                  
END_PROGRAM

PROGRAM prg_Hmi_FrameMiniPCMenu
  VAR
    iSelectionFrameMiniPCMenu : INT;
    xTB_Home : BOOL;
  END_VAR

                    IF xTB_Home THEN
	xTB_Home := FALSE;
	iSelectionFrameMiniPCMenu := 0;
END_IF
                  
END_PROGRAM

PROGRAM prg_Hmi_ManagerMiniPC
  VAR
    sDescriptionBar : STRING(255) := 'Stato Gestore CubeOS:';
    sStatusMessage : STRING(255);
  END_VAR

                    // IF visuElems.CURRENTLANGUAGE = 'it' THEN
// 	sDescriptionBar := 'Gestore MiniPC:';
// ELSE
// 	sDescriptionBar := 'MiniPC manager:';
// END_IF

// sStatusMessage := GVL.g_PM_HMI_StatusMessages.sMiniPCManager;
                  
END_PROGRAM

PROGRAM prg_Hmi_InterfaceSetting
  VAR
    sDescriptionBar : STRING(255) := 'Stato impostazioni:';
    sStatusMessage : STRING(255);
  END_VAR

                    
                  
END_PROGRAM

PROGRAM prg_Hmi_RobotMenu
  VAR
    sDescriptionBar : STRING(255) := 'Stato Robot:';
    sStatusMessage : STRING(255);
    xTB_Refresh : BOOL;
    xDIS_Refresh : BOOL;
    sWebServerURL : STRING(255) := 'http://192.168.1.232:3000';
    xShowWebServerPage : BOOL := TRUE;
    sTestImageBitmap : STRING(255) := '/home/andrea/temp/history/detection_2023-03-31-09:36:17.png';
  END_VAR

                    xDIS_Refresh := xShowWebServerPage;
IF xTB_Refresh THEN
	xTB_Refresh := FALSE;
	xShowWebServerPage := TRUE;
END_IF
                  
END_PROGRAM

PROGRAM prg_Hmi_FrameRobotMenu
  VAR
    iSelectionFrameRobotMenu : INT;
    xTB_Home : BOOL;
  END_VAR

                    IF xTB_Home THEN
	xTB_Home := FALSE;
	iSelectionFrameRobotMenu := 0;
END_IF
                  
END_PROGRAM

PROGRAM prg_Hmi_ErrorFrame
  VAR
    iSelectionFrame : INT;
    sStatusMessage : STRING(255);
    sDescriptionBar : STRING(255);
  END_VAR

                    
                  
END_PROGRAM

PROGRAM prg_Hmi_Application
  VAR
    ROSInterface_01 : ros_interface_struct_t;
    xTB_Run_01 : BOOL;
    xDIS_Run_01 : BOOL;
    eROSProcessState_01 : process_code_enum_t;
    ROSInterface_02 : ros_interface_struct_t;
    xTB_Run_02 : BOOL;
    xDIS_Run_02 : BOOL;
    eROSProcessState_02 : process_code_enum_t;
    diProcessCode_01 : DINT;
    dwColorProcessState_01 : DWORD;
    eProcessState_01 : process_code_enum_t;
    dwFontColorID_01 : DWORD;
    diProcessCode_02 : DINT;
    dwColorProcessState_02 : DWORD;
    eProcessState_02 : process_code_enum_t;
    dwFontColorID_02 : DWORD;
    eDoosanRobotState : doosan_robot_state_enum_t;
    dwColorDoosanState : DWORD;
    xDIS_Run : BOOL;
    eDoosanRobotState_2 : doosan_robot_state_enum_t;
    dwColorDoosanState_2 : DWORD;
    xCommunicationError_2 : BOOL;
    xCommunicationError : BOOL;
    xINVIS_CommErr : BOOL;
    xDangerBlinkRed : BOOL;
    xEnableDangerBlinking : BOOL;
    xDangerBlinkRed_2 : BOOL;
    xINVIS_CommErr_2 : BOOL;
    sDescriptionBar : STRING(255) := 'Stato applicazione:';
    sStatusMessage : STRING(255);
  END_VAR

                    // IF visuElems.CURRENTLANGUAGE = 'it' THEN

ROSInterface_01 := prgROS.ROSInterface_01;
xTB_Run_01 := TO_BOOL(ROSInterface_01.Codesys2ROS.Published.run);
eROSProcessState_01 := ROSInterface_01.ROS2Codesys.eProcessState;
(*--------------------------------*)
ROSInterface_02 := prgROS.ROSInterface_02;
xTB_Run_02 := TO_BOOL(ROSInterface_02.Codesys2ROS.Published.run);
eROSProcessState_02 := ROSInterface_02.ROS2Codesys.eProcessState;

(*======================================================*)
diProcessCode_01 := prgROS.ROSInterface_01.ROS2Codesys.Subscripted.process_code;
eProcessState_01 := prgROS.ROSInterface_01.ROS2Codesys.eProcessState;

IF diProcessCode_01 < 0 THEN
	dwColorProcessState_01 := GVL_Constants.gc_dwRed;
ELSE
	dwColorProcessState_01 := GVL_Constants.gc_dwWhite;
END_IF

CASE eProcessState_01 OF
	process_code_enum_t.pcode_Error:
		dwFontColorID_01 := GVL_Constants.gc_dwRed;
	ELSE
		dwFontColorID_01 := GVL_Constants.gc_dwWhite;
END_CASE
(*======================================================*)
diProcessCode_02 := prgROS.ROSInterface_02.ROS2Codesys.Subscripted.process_code;
eProcessState_02 := prgROS.ROSInterface_02.ROS2Codesys.eProcessState;

IF diProcessCode_02 < 0 THEN
	dwColorProcessState_02 := GVL_Constants.gc_dwRed;
ELSE
	dwColorProcessState_02 := GVL_Constants.gc_dwWhite;
END_IF

CASE eProcessState_02 OF
	process_code_enum_t.pcode_Error:
		dwFontColorID_02 := GVL_Constants.gc_dwRed;
	ELSE
		dwFontColorID_02 := GVL_Constants.gc_dwWhite;
END_CASE

(**)

eDoosanRobotState := prgEIPMapping.DoosanState.eRobotState; //12/01/2023
CASE eDoosanRobotState OF
	doosan_robot_state_enum_t.EmergencyStop, doosan_robot_state_enum_t.SafeOff, doosan_robot_state_enum_t.BackdriveHold:
		dwColorDoosanState := GVL_Constants.gc_dwRed;
	doosan_robot_state_enum_t.StandaloneRunning:
		dwColorDoosanState := GVL_Constants.gc_dwGreen;
	ELSE
		dwColorDoosanState := GVL_Constants.gc_dwWhite;
END_CASE

xCommunicationError := prgEIPMapping.xCommunicationError;
IF xCommunicationError THEN
	xDangerBlinkRed := xEnableDangerBlinking AND prg_HMI_MainFrame.METH_GetBlinkSync_Slow();
ELSE
	xDangerBlinkRed := FALSE;
END_IF
IF xCommunicationError THEN
	xINVIS_CommErr := NOT prg_HMI_MainFrame.METH_GetBlinkSync_Fast();
ELSE
	xINVIS_CommErr := TRUE;
END_IF
// xDIS_Run := 
// 	(
// 		eDoosanRobotState = doosan_robot_state_enum_t.EmergencyStop 
// 		OR eDoosanRobotState = doosan_robot_state_enum_t.SafeOff 
// 		OR eDoosanRobotState = doosan_robot_state_enum_t.BackdriveHold
// 		OR prg_Hmi_RobotControl.eAdapterState <> IoDrvEtherNetIP.DEVICE_STATE.RUNNING
// 	) AND NOT METH_IsGazelle()
// ;

eDoosanRobotState_2 := prgEIPMapping.DoosanState_2.eRobotState; //12/01/2023
CASE eDoosanRobotState_2 OF
	doosan_robot_state_enum_t.EmergencyStop, doosan_robot_state_enum_t.SafeOff, doosan_robot_state_enum_t.BackdriveHold:
		dwColorDoosanState_2 := GVL_Constants.gc_dwRed;
	doosan_robot_state_enum_t.StandaloneRunning:
		dwColorDoosanState_2 := GVL_Constants.gc_dwGreen;
	ELSE
		dwColorDoosanState_2 := GVL_Constants.gc_dwWhite;
END_CASE

xCommunicationError_2 := prgEIPMapping.xCommunicationError_2;
IF xCommunicationError_2 THEN
	xDangerBlinkRed_2 := xEnableDangerBlinking AND prg_HMI_MainFrame.METH_GetBlinkSync_Slow();
ELSE
	xDangerBlinkRed_2 := FALSE;
END_IF
IF xCommunicationError_2 THEN
	xINVIS_CommErr_2 := NOT prg_HMI_MainFrame.METH_GetBlinkSync_Fast();
ELSE
	xINVIS_CommErr_2 := TRUE;
END_IF

                  

METHOD METH_IsGazelle : BOOL
                          METH_IsGazelle := prgMain.sHostName = 'gazelle';
                        
END_METHOD

METHOD METH_ToggleRun_01 : BOOL
  VAR
    xCurrentValue : BOOL;
    xVal : BOOL;
  END_VAR
                          xCurrentValue := TO_BOOL(prgROS.ROSInterface_01.Codesys2ROS.Published.run);
xVal := prgROS.METH_SetRun_01(xValue := NOT xCurrentValue);

METH_ToggleRun_01 := xVal;
                        
END_METHOD

METHOD METH_ToggleRun_02 : BOOL
  VAR
    xCurrentValue : BOOL;
    xVal : BOOL;
  END_VAR
                          xCurrentValue := TO_BOOL(prgROS.ROSInterface_02.Codesys2ROS.Published.run);
xVal := prgROS.METH_SetRun_02(xValue := NOT xCurrentValue);

METH_ToggleRun_02 := xVal;
                        
END_METHOD
END_PROGRAM

(* Implicitly generated code : DO NOT EDIT *)
{attribute 'check_bounds'}
{attribute 'no_check'}
FUNCTION CheckBounds : DINT
  VAR_INPUT
    index : DINT;
    lower : DINT;
    upper : DINT;
  END_VAR

                    // Implicitly generated code: Only an implementation suggestion
IF  index < lower THEN
	CheckBounds := lower;
ELSIF  index > upper THEN
	CheckBounds := upper;
ELSE  
	CheckBounds := index;
END_IF

(*It is also possible to set a breakpoint, log messages or e.g. to halt on an exception:
Add CmpApp.library, SysExcept.library and SysTypes2_Itf as newest.
Declaration:
VAR
    _pApp : POINTER TO CmpApp.APPLICATION;
    _result   : SysTypes.RTS_IEC_RESULT;
END_VAR

Implementation:
_pApp := AppGetCurrent(pResult:=_result);
IF  index < lower THEN
        CheckBounds := lower;
        IF _pApp <> 0 THEN
                AppGenerateException(pApp:=_pApp, ulException:=RtsExceptions.RTSEXCPT_ARRAYBOUNDS);
        END_IF
ELSIF  index > upper THEN
        CheckBounds := upper;
        IF _pApp <> 0 THEN
                AppGenerateException(pApp:=_pApp,   ulException:=RtsExceptions.RTSEXCPT_ARRAYBOUNDS);
        END_IF
ELSE  
        CheckBounds := index;
END_IF
*)

                  
END_FUNCTION

PROGRAM prgLinuxCommand
  VAR
    xTB_LinuxCommandTest : BOOL;
    xTB_NodeList : BOOL;
    diProcessExecuteResult : DINT;
    RTS_Result : SysProcess.RTS_IEC_RESULT;
    sCommand : STRING(255) := 'sudo pwd';
    sStdOutBuffer : STRING(1000);
    udiSizeStdOutBuffer : UDINT;
    iCounterFailure : INT;
    iCounterSuccess : INT;
    sLastStdOutResult : STRING(1000);
    sErrorMessage : STRING;
    xwCopySize : __XWORD;
    sPythonFile_Echo : STRING := 'echo.py';
    sPythonCommand_Echo : STRING(255) := 'CONCAT(c_sPythonExecute, sPythonFile_Echo)';
    sDestFullPath_Echo : STRING(255);
    sSourceFullPath_Echo : STRING(255);
    sBashFile_DockerActivate : STRING := 'launch_docker.sh';
    sBashCommand_DockerActivate : STRING(255) := 'CONCAT(c_sBashExecute, sBashFile_DockerActivate)';
    sDestFullPath_DockerActivate : STRING(255);
    sSourceFullPath_DockerActivate : STRING(255);
    sBashFile_RobinActivate : STRING := 'launch_remote_robin.sh';
    sBashCommand_RobinActivate : STRING(255) := 'CONCAT(c_sBashExecute, sBashFile_RobinActivate)';
    sDestFullPath_RobinActivate : STRING(255);
    sSourceFullPath_RobinActivate : STRING(255);
    xTB_ActivateDocker : BOOL;
    xTB_ActivateRobin : BOOL;
    sTestCommand : STRING(255) := 'sudo roscore';
    xTB_ShutdownMiniPC : BOOL;
    xDIS_Command : BOOL;
    xTB_RebootMiniPC : BOOL;
    xTB_StartDocker : BOOL;
    xTB_KillBehaviorTree : BOOL;
    xTB_StartBehaviorTree : BOOL;
    xTB_StopDocker : BOOL;
    xTB_ListDockers : BOOL;
    xListContainers : BOOL;
    sContainersAlive : STRING(1000);
    xTB_KillBoxDetection : BOOL;
    xTB_StartBoxDetection : BOOL;
    xTB_ReadFile : BOOL;
    RTS_FileCloseResult : RTS_IEC_RESULT;
    xListNodes : BOOL;
    sNodesAlive : STRING(255);
    TON_NodeList : TON;
    xTB_NodeListStartNode : BOOL;
    tTimeStart : TIME := TIME#3s0ms;
    TON_NodeListPolling : TON;
    xIsDockerDoosanStarted : BOOL;
    tPollingNodes : TIME := TIME#10s0ms;
    xTB_StartDoosanControl : BOOL;
    xTB_KillDoosanControl : BOOL;
    xTB_StartDoosanMover : BOOL;
    xTB_KillDoosanMover : BOOL;
    xIsDoosanControlStarted : BOOL;
    xIsDoosanMoverStarted : BOOL;
    xIsBoxRecognitionStarted : BOOL;
    xIsBehaviorStarted : BOOL;
    tPollingDocker : TIME := TIME#30s0ms;
    TON_DockerListPolling : TON;
    iStepStartAll : INT;
    xTB_StartAllNodes : BOOL;
    xNodeStartRequested : BOOL;
    xAllNodesDown : BOOL;  (* xTB_StopAllNodes: BOOL; *)
    xAllNodesAreUp : BOOL;
    xTB_START_DOOSAN : BOOL;
    xTB_STOP : BOOL;
    xTB_RECOVERY_TOOL_EMPTY : BOOL;
    xEnableListing : BOOL;
    xTB_RECOVERY_TOOL_BUNDLE : BOOL;
    xTB_RECOVERY_TOOL_STOP : BOOL;
    sCurrentDockerComposePath : STRING;
    xTB_START_BT01 : BOOL;
    xTB_START_BT02 : BOOL;
    xTB_STOP_BT01 : BOOL;
    xTB_STOP_BT02 : BOOL;
    xIsDockerBTStarted : BOOL;
    xIsDockerBTStarted01 : BOOL;
    xIsDockerBTStarted02 : BOOL;
  END_VAR
  VAR CONSTANT
    c_sDestPath : STRING := '/var/opt/codesys/';
    c_sSourcePath : STRING := '/var/opt/codesys/PlcLogic/Application/';
    c_sPythonExecute : STRING := 'sudo python ';
    c_sBashExecute : STRING := './';
    c_sDockerName : STRING := 'src-doosan';  (* philip_development //philip_devel-v2 //philip_development *)
    c_sDockerNameBT : STRING := 'src-behavior_tree';
    c_sDockerNameBT01 : STRING := 'src-behavior_tree1';
    c_sDockerNameBT02 : STRING := 'src-behavior_tree2';
    c_sDockerActivateFile : STRING := 'launch_docker.sh';
    c_sDockerComposePath_Gazelle : STRING := '/home/nicola/ros/philip_ws/src/';  (* 05/12/2022 *)
    c_sDockerComposePath_Cincoze : STRING := '/home/sysdesign/ros/philip_ws/src/';  (* 05/12/2022 *)
    c_sDockerComposePath_Esaware : STRING := '/home/sysdesign/ros/pallcube_ws/src/';  (* 05/12/2022 *)
  END_VAR

                    (*=======================================================*)
// MINI PC
ACT_MiniPC();

(*--------------------------------*)
// dockker list
ACT_DockerList();
(*--------------------------------*)
// docker compose command
ACT_Start();

ACT_Stop();

(*--------------------------------*)
// flags
xIsDoosanControlStarted := FIND(sNodesAlive, 'dsr01h2017') > 0;
xIsDoosanMoverStarted := FIND(sNodesAlive, 'doosan_mover') > 0;
xIsBoxRecognitionStarted := FIND(sNodesAlive, 'box_recognition') > 0;
xIsBehaviorStarted := FIND(sNodesAlive, 'behavior_tree') > 0;
(*--------------------------------*)
xDIS_Command := FALSE;
IF xTB_LinuxCommandTest THEN
	xTB_LinuxCommandTest := FALSE;
	xDIS_Command := TRUE; //06/12/2022
	
	sCommand := sTestCommand;
// 	sCommand := sPythonCommand_Echo;
	
	sErrorMessage := '';
	udiSizeStdOutBuffer := TO_UDINT(XSIZEOF(sStdOutBuffer));
	SysMem.SysMemSet(pDest := ADR(sStdOutBuffer), udiCount := XSIZEOF(sStdOutBuffer), udiValue := 0);
	
	diProcessExecuteResult := SysProcess.SysProcessExecuteCommand2(
		pszCommand := sCommand,
		pResult := ADR(RTS_Result),
		pszStdOut := sStdOutBuffer,
		udiStdOutLen := udiSizeStdOutBuffer
	);
	
	IF RTS_Result = CmpErrors.Errors.ERR_OK THEN
		iCounterSuccess := (iCounterSuccess + 1) MOD 16#7FFF;
		IF diProcessExecuteResult > 0 THEN // there is something to read
			sLastStdOutResult := sStdOutBuffer;
		END_IF
		IF xListContainers THEN
			xListContainers := FALSE;
			sContainersAlive := sStdOutBuffer;
		END_IF
		IF xListNodes THEN
			xListNodes := FALSE;
			sNodesAlive := sStdOutBuffer;
		END_IF
	ELSE
		sErrorMessage := METH_GetErrorMessage(udiResult := RTS_Result);
		iCounterFailure := (iCounterFailure + 1) MOD 16#7FFF;
		IF xListNodes THEN
			xListNodes := FALSE;
			sNodesAlive := '';
		END_IF
	END_IF
	
	xDIS_Command := FALSE; //06/12/2022
END_IF
(*=======================================================*)
                  

ACTION ACT_MiniPC:
                        IF xTB_ShutdownMiniPC OR GVL.g_xShutdownMiniPC THEN
	GVL.g_xShutdownMiniPC := FALSE;
	xTB_ShutdownMiniPC := FALSE;
	sTestCommand := 'sudo shutdown -h now';
	xTB_LinuxCommandTest := TRUE;
END_IF
IF xTB_RebootMiniPC THEN
	xTB_RebootMiniPC := FALSE;
	sTestCommand := 'sudo reboot';
	xTB_LinuxCommandTest := TRUE;
END_IF
                      
END_ACTION

ACTION ACT_DockerList:
                        // DOCKER list
TON_DockerListPolling(IN := xEnableListing, PT := tPollingDocker);
IF TON_DockerListPolling.Q THEN
	TON_DockerListPolling(IN := FALSE);
	xTB_ListDockers := TRUE;
END_IF
IF xTB_ListDockers OR GVL.g_xListDockers THEN
	GVL.g_xListDockers := FALSE;
	xTB_ListDockers := FALSE;
	sTestCommand := 'docker container ls';
	xTB_LinuxCommandTest := TRUE;
	xListContainers := TRUE;
END_IF

xIsDockerDoosanStarted := STU.StrFindA(pst1 := ADR(sContainersAlive), pst2 := ADR(c_sDockerName), uiSearchStart := 0) > 0;
xIsDockerBTStarted := STU.StrFindA(pst1 := ADR(sContainersAlive), pst2 := ADR(c_sDockerNameBT), uiSearchStart := 0) > 0;
xIsDockerBTStarted01 := STU.StrFindA(pst1 := ADR(sContainersAlive), pst2 := ADR(c_sDockerNameBT01), uiSearchStart := 0) > 0;
xIsDockerBTStarted02 := STU.StrFindA(pst1 := ADR(sContainersAlive), pst2 := ADR(c_sDockerNameBT02), uiSearchStart := 0) > 0;
TON_NodeListPolling(IN := xIsDockerDoosanStarted AND xEnableListing, PT := tPollingNodes);
IF TON_NodeListPolling.Q THEN
	TON_NodeListPolling(IN := FALSE);
	xTB_NodeList := TRUE;
END_IF
(*===============================================*)
// LIST
IF xTB_NodeList THEN
	xTB_NodeList := FALSE;
// 	sTestCommand := './launch_docker.sh';
	sTestCommand := '';
// 	sTestCommand := 'docker exec ';
// 	sTestCommand := CONCAT(sTestCommand, c_sDockerName);
// 	sTestCommand := CONCAT(sTestCommand, ' bash -c $'source devel/setup.bash; rosnode list$'');
	sTestCommand := 'bash -c $'source /opt/ros/noetic/setup.bash; rosnode list$'';
	xTB_LinuxCommandTest := TRUE;
	xListNodes := TRUE;
END_IF
(*--------------------------------*)
                      
END_ACTION

ACTION ACT_Start:
                        // DOOSAN
IF xTB_START_DOOSAN OR GVL.g_xNODES_START THEN // START DOOSAN
	xTB_START_DOOSAN := FALSE;
	GVL.g_xNODES_START := FALSE;
	sTestCommand := '';
	sCurrentDockerComposePath := METH_GetDockerComposePath();
	sTestCommand := CONCAT('docker compose -f ', CONCAT(sCurrentDockerComposePath, 'docker-compose.yml up -d doosan'));
	// 		sTestCommand := 'docker compose -f /home/nicola/ros/philip_ws/src/docker-compose.devel.yml up -d';
	// 	sTestCommand := 'bash /home/sysdesign/philip.sh start';
	xTB_LinuxCommandTest := TRUE;
END_IF

// BT
IF xTB_START_BT01 THEN // START DOOSAN
	xTB_START_BT01 := FALSE;
	sTestCommand := '';
	sCurrentDockerComposePath := METH_GetDockerComposePath();
	sTestCommand := CONCAT('docker compose -f ', CONCAT(sCurrentDockerComposePath, 'docker-compose.yml up -d behavior_tree1'));
	// 		sTestCommand := 'docker compose -f /home/nicola/ros/philip_ws/src/docker-compose.devel.yml up -d';
	// 	sTestCommand := 'bash /home/sysdesign/philip.sh start';
	xTB_LinuxCommandTest := TRUE;
END_IF

IF xTB_START_BT02 THEN // START DOOSAN
	xTB_START_BT02 := FALSE;
	sTestCommand := '';
	sCurrentDockerComposePath := METH_GetDockerComposePath();
	sTestCommand := CONCAT('docker compose -f ', CONCAT(sCurrentDockerComposePath, 'docker-compose.yml up -d behavior_tree2'));
	// 		sTestCommand := 'docker compose -f /home/nicola/ros/philip_ws/src/docker-compose.devel.yml up -d';
	// 	sTestCommand := 'bash /home/sysdesign/philip.sh start';
	xTB_LinuxCommandTest := TRUE;
END_IF
                      
END_ACTION

ACTION ACT_Stop:
                        IF xTB_STOP OR GVL.g_xNODES_STOP THEN
	xTB_STOP := FALSE;
	GVL.g_xNODES_STOP := FALSE;
	sTestCommand := '';
	sCurrentDockerComposePath := METH_GetDockerComposePath();
	sTestCommand := CONCAT('docker compose -f ', CONCAT(sCurrentDockerComposePath, 'docker-compose.yml down')); //23/01/2023: perche non STOP?
	// 		sTestCommand := 'docker compose -f /home/nicola/ros/philip_ws/src/docker-compose.devel.yml down';
// 		sTestCommand := 'bash /home/sysdesign/philip.sh stop';
	xTB_LinuxCommandTest := TRUE;
END_IF


IF xTB_STOP_BT01 THEN // START DOOSAN
	xTB_STOP_BT01 := FALSE;
	sTestCommand := '';
	sCurrentDockerComposePath := METH_GetDockerComposePath();
	sTestCommand := CONCAT('docker compose -f ', CONCAT(sCurrentDockerComposePath, 'docker-compose.yml stop behavior_tree1'));
	// 		sTestCommand := 'docker compose -f /home/nicola/ros/philip_ws/src/docker-compose.devel.yml up -d';
	// 	sTestCommand := 'bash /home/sysdesign/philip.sh start';
	xTB_LinuxCommandTest := TRUE;
END_IF

IF xTB_STOP_BT02 THEN // START DOOSAN
	xTB_STOP_BT02 := FALSE;
	sTestCommand := '';
	sCurrentDockerComposePath := METH_GetDockerComposePath();
	sTestCommand := CONCAT('docker compose -f ', CONCAT(sCurrentDockerComposePath, 'docker-compose.yml stop behavior_tree2'));
	// 		sTestCommand := 'docker compose -f /home/nicola/ros/philip_ws/src/docker-compose.devel.yml up -d';
	// 	sTestCommand := 'bash /home/sysdesign/philip.sh start';
	xTB_LinuxCommandTest := TRUE;
END_IF
                      
END_ACTION

METHOD METH_GetErrorMessage : STRING(255)
  VAR_INPUT
    udiResult : SysProcess.RTS_IEC_RESULT;
  END_VAR
  VAR
    sRes : STRING(255);
  END_VAR
                          CASE udiResult OF
	CmpErrors.Errors.ERR_PARAMETER:
		sRes := 'Some null input parameter';
	CmpErrors.Errors.ERR_NO_ACCESS_RIGHTS:
		sRes := 'Not allowed';
	CmpErrors.Errors.ERR_FAILED:
		sRes := 'Internal error';
	ELSE
		sRes := 'Error';
END_CASE

METH_GetErrorMessage := sRes;
                        
END_METHOD

METHOD METH_GetDockerComposePath : STRING
  VAR
    sRes : STRING;
  END_VAR
                          IF prgMAIN.sHostName = 'gazelle' OR prgMAIN.sHostName = 'esaware' THEN
	sRes := c_sDockerComposePath_Esaware;
ELSE
	sRes := c_sDockerComposePath_Cincoze;
END_IF

METH_GetDockerComposePath := sRes;
                        
END_METHOD

METHOD METH_StartDoosanDocker
                          xTB_START_DOOSAN := TRUE;
                        
END_METHOD

METHOD METH_StartBT01
                          xTB_START_BT01 := TRUE;
                        
END_METHOD

METHOD METH_StartBT02
                          xTB_START_BT02 := TRUE;
                        
END_METHOD

METHOD METH_StopAllDockers
                          xTB_STOP := TRUE;
                        
END_METHOD

METHOD METH_ShutdownMiniPC
                          xTB_ShutdownMiniPC := TRUE;
                        
END_METHOD

METHOD METH_RebootMiniPC
                          xTB_RebootMiniPC := TRUE;
                        
END_METHOD

METHOD METH_ListDockers
                          xTB_ListDockers := TRUE;
                        
END_METHOD

METHOD METH_IsDockerDoosanActive : BOOL
                          METH_IsDockerDoosanActive := xIsDockerDoosanStarted;

                        
END_METHOD

METHOD METH_IsDockerBTActive : BOOL
                          METH_IsDockerBTActive := xIsDockerBTStarted;

                        
END_METHOD

METHOD METH_IsDockerBTActive_01 : BOOL
                          METH_IsDockerBTActive_01 := xIsDockerBTStarted01;

                        
END_METHOD

METHOD METH_IsDockerBTActive_02 : BOOL
                          METH_IsDockerBTActive_02 := xIsDockerBTStarted02;

                        
END_METHOD

METHOD METH_StopBT01
                          xTB_STOP_BT01 := TRUE;
                        
END_METHOD

METHOD METH_StopBT02
                          xTB_STOP_BT02 := TRUE;
                        
END_METHOD
END_PROGRAM

PROGRAM prgEIPMapping
  VAR
    bRobotState : BYTE;
    bRobotFlags : BYTE;
    DoosanState : doosan_state_struct_t;  (* 16/12/2022 *)
    xCommunicationError : BOOL;
    xAirAspriration : BOOL;
    bRobotState_2 : BYTE;
    bRobotFlags_2 : BYTE;
    DoosanState_2 : doosan_state_struct_t;  (* 16/12/2022 *)
    xCommunicationError_2 : BOOL;
    TON_Dead_2 : TON;
    Doosan_EIP : doosan_t;
    Doosan_EIP_2 : doosan_t;
    udiRobotState : UDINT;
    xErrorArea : BOOL;
    TON_Dead : TON;  (* eProposedDoosanArea : PM_areas_enum_t; *)
    tDead : TIME := TIME#5s0ms;
    xInit : BOOL := TRUE;
    pxTurnOn : POINTER TO BOOL;
    xEthercatError : BOOL;
    xStartDocker : BOOL;
    xRecoveryZoneError : BOOL;
    xInRecoveryZone : BOOL;
  END_VAR

                    // EIP mask inputs
IO_Variables.g_Doosan_EIP.Cartesian := Doosan_EIP.Cartesian;
IO_Variables.g_Doosan_EIP.Joints := Doosan_EIP.Joints;
IO_Variables.g_Doosan_EIP.InfoRobot := Doosan_EIP.InfoRobot;

// eProposedDoosanArea := METH_GetArea(xError => xErrorArea, xIsAlive => IO_Variables.g_Doosan_EIP.xIsAlive); //20/10/2022: is alive
// IF NOT xErrorArea THEN
// 	IO_Variables.g_eDoosanArea := eProposedDoosanArea;
// ELSE
// 	IO_Variables.g_eDoosanArea := PM_areas_enum_t.UnknownArea;
// END_IF

xInRecoveryZone := METH_GetJointsLimitDanger(xError => xRecoveryZoneError); //07/12/2022

// 20/10/2022: automatically turn on doosan if
IO_Variables.g_Doosan_EIP.xIsAlive := prg_Hmi_RobotControl.eAdapterState = IoDrvEtherNetIP.DEVICE_STATE.RUNNING;//20/10/2022
xCommunicationError := NOT IO_Variables.g_Doosan_EIP.xIsAlive;
TON_Dead(IN := NOT IO_Variables.g_Doosan_EIP.xIsAlive, PT := tDead); //20/10/2022
GVL.g_xDoosanMayBeOff := TON_Dead.Q; //20/10/2022

IO_Variables.g_Doosan_EIP_2.xIsAlive := prg_Hmi_RobotControl2.eAdapterState = IoDrvEtherNetIP.DEVICE_STATE.RUNNING;//20/10/2022
xCommunicationError_2 := NOT IO_Variables.g_Doosan_EIP_2.xIsAlive;
TON_Dead_2(IN := NOT IO_Variables.g_Doosan_EIP_2.xIsAlive, PT := tDead); //20/10/2022
GVL.g_xDoosanMayBeOff_2 := TON_Dead_2.Q; //20/10/2022
// xEthercatError := 
// 	(prgMain.eEthercatState <> DED.BUS_STATE.RUNNING
// 	OR prgMain.eEthercatError <> DED.ERROR.NO_ERROR)
// // 	AND prgMain.xEthercatDiagnosisAvail //07/12/2022: commentato
// ; //24/10/2022: controllo ethercat prima di mandare segnale
// IF xInit THEN  
// 	IF IO_Variables.g_Doosan_EIP.xIsAlive THEN//20/10/2022
// 		xInit := FALSE;
// 		xStartDocker := TRUE; //28/10/2022: at startup also start docker
// 	ELSE  
// 		IF GVL.g_xDoosanMayBeOff AND NOT xEthercatError THEN //24/10/2022 //20/10/2022 
// // 			pxTurnOn := ADR(prg_Hmi_Home.xTB_TurnDoosanON);
// // 			pxTurnOn^ := TRUE;
// 			prg_Hmi_Home.METH_AskForDoosanOn();
// 			xInit := FALSE;
// 			xStartDocker := TRUE; //28/10/2022: at startup also start docker
// 		END_IF
// 	END_IF
// ELSIF xStartDocker THEN //28/10/2022 starts docker at startup
// 	IF IO_Variables.g_Doosan_EIP.xIsAlive THEN
// 		GVL.g_xNODES_START := TRUE;
// 		xStartDocker := FALSE;
// 	END_IF
// END_IF
(*--------------------------------------------------------------*)
//16/12/2022: flag per capire se stato robot è quel che voglio
DoosanState.eRobotState := bRobotState;
DoosanState.xSO_ServoOn := bRobotFlags.0;
DoosanState.xSS_SafetyStopped := bRobotFlags.1;
DoosanState.xES_EmergencyStopped := bRobotFlags.2;
DoosanState.xDTPB_DirectTeachButtonPressed := bRobotFlags.3;
DoosanState.xPBP_PowerButtonPressed := bRobotFlags.4;

DoosanState_2.eRobotState := bRobotState_2;
DoosanState_2.xSO_ServoOn := bRobotFlags_2.0;
DoosanState_2.xSS_SafetyStopped := bRobotFlags_2.1;
DoosanState_2.xES_EmergencyStopped := bRobotFlags_2.2;
DoosanState_2.xDTPB_DirectTeachButtonPressed := bRobotFlags_2.3;
DoosanState_2.xPBP_PowerButtonPressed := bRobotFlags_2.4;



                  

(* This method proposes an area, but if more then one is found, then it throws an error *)
METHOD METH_GetArea : PM_areas_enum_t
  VAR_OUTPUT
    xError : BOOL;
    xIsAlive : BOOL;  (* 20/10/2022 *)
  END_VAR
  VAR
    eRes : PM_areas_enum_t;
    aHome_WindowX : ARRAY[0..1] OF REAL := [(-640.0 - 200), (-640.0 + 200.0)];
    aHome_WindowY : ARRAY[0..1] OF REAL := [(-210.0 - 200), (-210.0 + 200)];
    aHome_WindowZ : ARRAY[0..1] OF REAL := [700.0, 1100.0];
    xInHomeArea : BOOL;
    aLoadCube_WindowX : ARRAY[0..1] OF REAL := [0.0, 0.0];
    aLoadCube_WindowY : ARRAY[0..1] OF REAL := [0.0, 0.0];
    aLoadCube_WindowZ : ARRAY[0..1] OF REAL := [0.0, 0.0];
    xInLoadCubeArea : BOOL;
    aPallet_WindowX : ARRAY[0..1] OF REAL := [0.0, 0.0];
    aPallet_WindowY : ARRAY[0..1] OF REAL := [0.0, 0.0];
    aPallet_WindowZ : ARRAY[0..1] OF REAL := [0.0, 0.0];
    xInPalletArea : BOOL;
    aSenzani_WindowX : ARRAY[0..1] OF REAL := [0.0, 0.0];
    aSenzani_WindowY : ARRAY[0..1] OF REAL := [0.0, 0.0];
    aSenzani_WindowZ : ARRAY[0..1] OF REAL := [0.0, 0.0];
    xInSenzaniArea : BOOL;
    lrX : REAL;
    lrY : REAL;
    lrZ : REAL;
    lrA : REAL;
    lrB : REAL;
    lrC : REAL;
    xConflict : BOOL;
    xAllZero : BOOL;
    xAllZeroJoints : BOOL;
  END_VAR
                          lrX := IO_Variables.g_Doosan_EIP.Cartesian.x;
lrY := IO_Variables.g_Doosan_EIP.Cartesian.y;
lrZ := IO_Variables.g_Doosan_EIP.Cartesian.z;
lrA := IO_Variables.g_Doosan_EIP.Cartesian.A;
lrB := IO_Variables.g_Doosan_EIP.Cartesian.B;
lrC := IO_Variables.g_Doosan_EIP.Cartesian.C;

xAllZero := lrX = 0.0 AND lrY = 0.0 AND lrZ = 0.0 AND lrA = 0.0 AND lrB = 0.0 AND lrC = 0.0;
xAllZeroJoints := 
	IO_Variables.g_Doosan_EIP.Joints.j1 = 0.0
	AND IO_Variables.g_Doosan_EIP.Joints.j2 = 0.0
	AND IO_Variables.g_Doosan_EIP.Joints.j3 = 0.0
	AND IO_Variables.g_Doosan_EIP.Joints.j4 = 0.0
	AND IO_Variables.g_Doosan_EIP.Joints.j5 = 0.0
	AND IO_Variables.g_Doosan_EIP.Joints.j6 = 0.0
;

xInHomeArea := 
	(lrX >= aHome_WindowX[0] AND lrX <= aHome_WindowX[1])
	AND (lrY >= aHome_WindowY[0] AND lrY <= aHome_WindowY[1])
	AND (lrZ >= aHome_WindowZ[0] AND lrZ <= aHome_WindowZ[1])
;

// 13/01/2023:  in load cube area for turning off
aLoadCube_WindowX := aHome_WindowX;
aLoadCube_WindowY := aHome_WindowY;
aHome_WindowZ[0] := 200.0;
aHome_WindowZ[1] := aHome_WindowZ[0];
xInLoadCubeArea := 
	(lrX >= aLoadCube_WindowX[0] AND lrX <= aLoadCube_WindowX[1])
	AND (lrY >= aLoadCube_WindowY[0] AND lrY <= aLoadCube_WindowY[1])
	AND (lrZ >= aLoadCube_WindowZ[0] AND lrZ <= aLoadCube_WindowZ[1])
;

xInPalletArea := 
	(lrX >= aPallet_WindowX[0] AND lrX <= aPallet_WindowX[1])
	AND (lrY >= aPallet_WindowY[0] AND lrY <= aPallet_WindowY[1])
	AND (lrZ >= aPallet_WindowZ[0] AND lrZ <= aPallet_WindowZ[1])
;

xInSenzaniArea := 
	(lrX >= aSenzani_WindowX[0] AND lrX <= aSenzani_WindowX[1])
	AND (lrY >= aSenzani_WindowY[0] AND lrY <= aSenzani_WindowY[1])
	AND (lrZ >= aSenzani_WindowZ[0] AND lrZ <= aSenzani_WindowZ[1])
;

xConflict := TO_INT(xInHomeArea) + TO_INT(xInLoadCubeArea) + TO_INT(xInPalletArea) + TO_INT(xInSenzaniArea) > 1;

xError := xConflict OR xAllZero;

IF xInHomeArea THEN
	eRes := PM_areas_enum_t.HomeArea;
ELSIF xInLoadCubeArea THEN
	eRes := PM_areas_enum_t.LoadCubeArea;
ELSIF xInPalletArea THEN
	eRes := PM_areas_enum_t.PalletArea;
ELSIF xInSenzaniArea THEN
	eRes := PM_areas_enum_t.SenzaniArea;
ELSE
	eRes := PM_areas_enum_t.UnknownArea;
END_IF

xIsAlive := NOT (xAllZero AND xAllZeroJoints);

METH_GetArea := eRes;
                        
END_METHOD

(* This method proposes an area, but if more then one is found, then it throws an error *)
METHOD METH_GetJointsLimitDanger : BOOL
  VAR_OUTPUT
    xError : BOOL;
  END_VAR
  VAR
    xAllZeroJoints : BOOL;
    iInd : INT;
    iMaxInd : INT := 5;
    rJointVal : REAL;
    rAbsLimit : REAL;
    rTolerance : REAL;
    axJointsDanger : ARRAY[0..5] OF BOOL;
    xRes : BOOL;
  END_VAR
                          
xAllZeroJoints := 
	IO_Variables.g_Doosan_EIP.Joints.j1 = 0.0
	AND IO_Variables.g_Doosan_EIP.Joints.j2 = 0.0
	AND IO_Variables.g_Doosan_EIP.Joints.j3 = 0.0
	AND IO_Variables.g_Doosan_EIP.Joints.j4 = 0.0
	AND IO_Variables.g_Doosan_EIP.Joints.j5 = 0.0
	AND IO_Variables.g_Doosan_EIP.Joints.j6 = 0.0
;
FOR iInd := 0 TO iMaxInd DO
	CASE iInd OF
		0: 
			rJointVal := IO_Variables.g_Doosan_EIP.Joints.j1;
			rAbsLimit := TO_REAL(ABS(360.0));
		1:
			rJointVal := IO_Variables.g_Doosan_EIP.Joints.j2;
			rAbsLimit := TO_REAL(ABS(360.0));
		2:
			rJointVal := IO_Variables.g_Doosan_EIP.Joints.j2;
			rAbsLimit := TO_REAL(ABS(360.0));
		3:
			rJointVal := IO_Variables.g_Doosan_EIP.Joints.j2;
			rAbsLimit := TO_REAL(ABS(360.0));
		4:
			rJointVal := IO_Variables.g_Doosan_EIP.Joints.j2;
			rAbsLimit := TO_REAL(ABS(90.0));
		5:
			rJointVal := IO_Variables.g_Doosan_EIP.Joints.j2;
			rAbsLimit := TO_REAL(ABS(360.0));
	END_CASE
	axJointsDanger[iInd] := rJointVal <= -rAbsLimit OR rJointVal >= rAbsLimit;
	xRes := xRes OR axJointsDanger[iInd];
END_FOR


xError := xAllZeroJoints;

METH_GetJointsLimitDanger := xRes;
                        
END_METHOD

METHOD METH_IsDoosanServoOn : BOOL
  VAR_INPUT
    DoosanState : doosan_state_struct_t;
  END_VAR
                          METH_IsDoosanServoOn := DoosanState.xSO_ServoOn;
                        
END_METHOD

METHOD METH_IsDoosanReadyForManual : BOOL
  VAR_INPUT
    DoosanState : doosan_state_struct_t;
  END_VAR
                          METH_IsDoosanReadyForManual := DoosanState.eRobotState = doosan_robot_state_enum_t.ManualStandby;
                        
END_METHOD

METHOD METH_IsDoosanReadyForAuto : BOOL
  VAR_INPUT
    DoosanState : doosan_state_struct_t;
  END_VAR
                          METH_IsDoosanReadyForAuto := DoosanState.eRobotState = doosan_robot_state_enum_t.StandaloneStandby;
                        
END_METHOD

METHOD METH_IsDoosanSafeOff : BOOL
  VAR_INPUT
    DoosanState : doosan_state_struct_t;
  END_VAR
                          METH_IsDoosanSafeOff := DoosanState.eRobotState = doosan_robot_state_enum_t.SafeOff;
                        
END_METHOD

METHOD METH_IsDoosanTurnedOff : BOOL
  VAR_INPUT
    eAdapterState : IoDrvEtherNetIP.DEVICE_STATE;
  END_VAR
                          METH_IsDoosanTurnedOff := prg_Hmi_RobotControl.eAdapterState = IoDrvEtherNetIP.DEVICE_STATE.NOT_FOUND;
                        
END_METHOD
END_PROGRAM

PROGRAM prg_Hmi_AskedPose
  VAR
    xINVIS_JointsResults : BOOL := TRUE;
    xINVIS_CartResults : BOOL := TRUE;
    arValues : ARRAY[0..7] OF REAL;
    xTB_Convert : BOOL;
    diLengthValues : DINT;
    sValues : STRING(255);
    diInd : DINT;
    sCurrentValue : STRING(255);
    iStartPos : INT;
    iLength : INT;
    uiStartSearch : UINT;
    iFindINd : INT;
    iIndValues : INT;
    eInputType : pose_type_t;
    xDIS_EnableConversion : BOOL;
    iMinInputType : INT := ANY_TO_INT(pose_type_t.JointDegrees);
    iMaxInputType : INT := ANY_TO_INT(pose_type_t.Cart_m_quat);
    xConvertToJointRadians : BOOL;
    xConvertToJointDegrees : BOOL;
    xConvertFromZYZ : BOOL;
    xConvertFromRPY : BOOL;
    xConvertFromQuat : BOOL;
    iIndJoints : INT;
    xIgnoreCart : BOOL;
    udiAuxBufferSize : UDINT;
    sZYZ : STRING(255);
    rA : REAL;
    rB : REAL;
    rC : REAL;
    lrA : LREAL;
    lrB : LREAL;
    lrC : LREAL;
    sDescriptionBar : STRING(255);
    sStatusBar : STRING(255);
    sjAux : STRING;  (* - *)
    sStringJointPos : STRING;
    scAux : STRING;  (* - *)
    sStringCartPos : STRING;
    sQuaternion : STRING(255);
    lrRoll : LREAL;
    lrPitch : LREAL;
    lrYaw : LREAL;
    xToRPY : BOOL;
    rRoll : REAL;
    rPitch : REAL;
    rYaw : REAL;
    rXmm : REAL;
    rYmm : REAL;
    rZmm : REAL;
    sRPY : STRING(255);
    xIsRot : BOOL;
    arJointsInRadians : ARRAY[0..5] OF REAL;
    arJointsInDegrees : ARRAY[0..5] OF REAL;
    arCartZYZ : ARRAY[0..5] OF REAL;
    arCartQuat : ARRAY[0..5] OF REAL;
    arCartRPY : ARRAY[0..5] OF REAL;
    xTB_ParseString : BOOL;
    Set_IP : BOOL;
    ipDosan : ARRAY[0..3] OF BYTE;
    deinfo : IoDrvEtherNetIP.DEVICE_INFO;
    errorDE : IoDrvEtherNetIP.DED.ERROR;
    a_ipDoosan : ARRAY[0..3] OF ARRAY[0..3] OF STRING := [['192', '168', '1', '70'], 3([4('')])];
    iIndexIP : INT := 1;  (* -Default impostato sul Doosan *)
    rXMeters : REAL;
    rYMeters : REAL;
    rZMeters : REAL;
    rQW : REAL;
    rQX : REAL;
    rQY : REAL;
    rQZ : REAL;
    mR : SM3M.SMC_Matrix3;
    xComputeRotMat : BOOL;
    q : SM3M.SMC_Quat;
    quat : SM3M.SMC_Quat;
    sAux : STRING(255);
    iBufferSize : INT;
    sJointsInRadians : STRING(255);
    sJointsInDegrees : STRING(255);
  END_VAR

                    IF xTB_ParseString OR xTB_Convert THEN
	xINVIS_CartResults := TRUE;
	xINVIS_JointsResults := TRUE;
	xConvertToJointRadians := FALSE;
	xConvertToJointDegrees := FALSE;
	xConvertFromQuat := FALSE;
	xConvertFromRPY := FALSE;
	xConvertFromZYZ := FALSE;
	
	xTB_ParseString := FALSE;
	SysMem.SysMemSet(pDest := ADR(arValues), udiCount := XSIZEOF(arValues), udiValue := 0);
	diLengthValues := STU.StrLenA(pstData := ADR(sValues));
	diInd := 0;
	iStartPos := 0;
	iLength := 0;
	iIndValues := 0;
	WHILE diInd < diLengthValues DO
		sCurrentValue := '';
		uiStartSearch := TO_UINT(diInd);
		iFindInd := STU.StrCaseFindA(pst1 := ADR(sValues), pst2 := ADR(';'), uiSearchStart := uiStartSearch);
		IF iFindInd > 0 THEN
			IF diInd = 0 THEN // first value
				iStartPos := 1;
			ELSE
				iStartPos := TO_INT(diInd);
			END_IF
			iLength := iFindInd - iStartPos;
			
			STU.StrMidA(
				pstResult := ADR(sCurrentValue),
				uiResultBufferSize := TO_UINT(XSIZEOF(sCurrentValue)),
				pst := ADR(sValues),
				uiInputBufferSize := TO_UINT(XSIZEOF(sValues)),
				iPosition := iStartPos,
				iLength := iLength
			);
			arValues[iIndValues] := STRING_TO_REAL(sCurrentValue);
			iIndValues := iIndValues + 1;
			
			diInd := TO_DINT(iFindInd + 1);
		ELSE
			IF iStartPos > 0 THEN // last value (no ;)
				iStartPos := TO_INT(diInd);
				iLength := TO_INT(diLengthValues) + 1 - iStartPos;
				STU.StrMidA(
					pstResult := ADR(sCurrentValue),
					uiResultBufferSize := TO_UINT(XSIZEOF(sCurrentValue)),
					pst := ADR(sValues),
					uiInputBufferSize := TO_UINT(XSIZEOF(sValues)),
					iPosition := iStartPos,
					iLength := iLength
				);
				
				arValues[iIndValues] := STRING_TO_REAL(sCurrentValue);
				iIndValues := iIndValues + 1;
				diInd := diLengthValues;
			END_IF
		END_IF
		
	END_WHILE
	
	IF iIndValues > 0 THEN
		CASE eInputType OF
			(*----------------------------------------*)
			// just convert to the other joint convention
			pose_type_t.JointDegrees:
				FOR iIndJoints := 0 TO 5 DO
					arJointsInDegrees[iIndJoints] := arValues[iIndJoints];
				END_FOR
				xConvertToJointRadians := TRUE;
				xINVIS_JointsResults := FALSE;
			pose_type_t.JointRadians:
				FOR iIndJoints := 0 TO 5 DO
					arJointsInRadians[iIndJoints] := arValues[iIndJoints];
				END_FOR
				xConvertToJointDegrees := TRUE;
				xINVIS_JointsResults := FALSE;
			(*----------------------------------------*)
			(*----------------------------------------*)
			// to rotation matrix, then write all three
			pose_type_t.Cart_mm_ZYZ:
				xConvertFromZYZ := TRUE;
				xINVIS_CartResults := FALSE;
			pose_type_t.Cart_mm_RPY:
				xConvertFromRPY := TRUE;
				xINVIS_CartResults := FALSE;
			pose_type_t.Cart_m_quat:
				xConvertFromQuat := TRUE;
				xINVIS_CartResults := FALSE;
			(*----------------------------------------*)
		END_CASE
	END_IF
END_IF




IF xTB_Convert THEN
	xTB_Convert := FALSE;
// 	ACT_ConcatCartPosString();
// 	ACT_ConcatJointPosString();
// 	
// 	ACT_Quaternions();
	
	ACT_JointsInRadians();
	ACT_JointsInDegrees();
	
	ACT_CartConvToMatrix();
	
END_IF












                  

ACTION ACT_RPY:
                        // RPY
iBufferSize := TO_INT(XSIZEOF(sRPY));
udiAuxBufferSize := TO_UDINT(XSIZEOF(sAux));
sRPY := '';

sAux := ''; //X
STU.StuSprintf(pstFormat := ADR('%5.1f'), pVarAdr := ADR(rXmm), udiVarType := __SYSTEM.TYPE_CLASS.TYPE_REAL, pBuffer := ADR(sAux), dwBufferSize := udiAuxBufferSize);
// sAux := TO_STRING(rXmm);
STU.StrConcatA(pstTo := ADR(sRPY), pstFrom := ADR(sAux), iBufferSize := iBufferSize);

STU.StrConcatA(pstTo := ADR(sRPY), pstFrom := ADR(';'), iBufferSize := iBufferSize);

sAux := ''; //Y
STU.StuSprintf(pstFormat := ADR('%5.1f'), pVarAdr := ADR(rYmm), udiVarType := __SYSTEM.TYPE_CLASS.TYPE_REAL, pBuffer := ADR(sAux), dwBufferSize := udiAuxBufferSize);
// sAux := TO_STRING(rYmm);
STU.StrConcatA(pstTo := ADR(sRPY), pstFrom := ADR(sAux), iBufferSize := iBufferSize);

STU.StrConcatA(pstTo := ADR(sRPY), pstFrom := ADR(';'), iBufferSize := iBufferSize);

sAux := ''; //Z
STU.StuSprintf(pstFormat := ADR('%5.1f'), pVarAdr := ADR(rZmm), udiVarType := __SYSTEM.TYPE_CLASS.TYPE_REAL, pBuffer := ADR(sAux), dwBufferSize := udiAuxBufferSize);
// sAux := TO_STRING(rZmm);
STU.StrConcatA(pstTo := ADR(sRPY), pstFrom := ADR(sAux), iBufferSize := iBufferSize);

STU.StrConcatA(pstTo := ADR(sRPY), pstFrom := ADR(';'), iBufferSize := iBufferSize);

sAux := ''; //roll
STU.StuSprintf(pstFormat := ADR('%3.1f'), pVarAdr := ADR(rRoll), udiVarType := __SYSTEM.TYPE_CLASS.TYPE_REAL, pBuffer := ADR(sAux), dwBufferSize := udiAuxBufferSize);
// sAux := TO_STRING(rRoll);
STU.StrConcatA(pstTo := ADR(sRPY), pstFrom := ADR(sAux), iBufferSize := iBufferSize);

STU.StrConcatA(pstTo := ADR(sRPY), pstFrom := ADR(';'), iBufferSize := iBufferSize);

sAux := ''; //pitch
STU.StuSprintf(pstFormat := ADR('%3.1f'), pVarAdr := ADR(rPitch), udiVarType := __SYSTEM.TYPE_CLASS.TYPE_REAL, pBuffer := ADR(sAux), dwBufferSize := udiAuxBufferSize);
// sAux := TO_STRING(rPitch);
STU.StrConcatA(pstTo := ADR(sRPY), pstFrom := ADR(sAux), iBufferSize := iBufferSize);

STU.StrConcatA(pstTo := ADR(sRPY), pstFrom := ADR(';'), iBufferSize := iBufferSize);

sAux := ''; //yaw
STU.StuSprintf(pstFormat := ADR('%3.1f'), pVarAdr := ADR(rYaw), udiVarType := __SYSTEM.TYPE_CLASS.TYPE_REAL, pBuffer := ADR(sAux), dwBufferSize := udiAuxBufferSize);
// sAux := TO_STRING(rYaw);
STU.StrConcatA(pstTo := ADR(sRPY), pstFrom := ADR(sAux), iBufferSize := iBufferSize);
                      
END_ACTION

ACTION ACT_ZYZ:
                        // RPY
iBufferSize := TO_INT(XSIZEOF(sZYZ));
udiAuxBufferSize := TO_UDINT(XSIZEOF(sAux));
sZYZ := '';

sAux := ''; //X
STU.StuSprintf(pstFormat := ADR('%5.1f'), pVarAdr := ADR(rXmm), udiVarType := __SYSTEM.TYPE_CLASS.TYPE_REAL, pBuffer := ADR(sAux), dwBufferSize := udiAuxBufferSize);
// sAux := TO_STRING(rXmm);
STU.StrConcatA(pstTo := ADR(sZYZ), pstFrom := ADR(sAux), iBufferSize := iBufferSize);

STU.StrConcatA(pstTo := ADR(sZYZ), pstFrom := ADR(';'), iBufferSize := iBufferSize);

sAux := ''; //Y
STU.StuSprintf(pstFormat := ADR('%5.1f'), pVarAdr := ADR(rYmm), udiVarType := __SYSTEM.TYPE_CLASS.TYPE_REAL, pBuffer := ADR(sAux), dwBufferSize := udiAuxBufferSize);
// sAux := TO_STRING(rYmm);
STU.StrConcatA(pstTo := ADR(sZYZ), pstFrom := ADR(sAux), iBufferSize := iBufferSize);

STU.StrConcatA(pstTo := ADR(sZYZ), pstFrom := ADR(';'), iBufferSize := iBufferSize);

sAux := ''; //Z
STU.StuSprintf(pstFormat := ADR('%5.1f'), pVarAdr := ADR(rZmm), udiVarType := __SYSTEM.TYPE_CLASS.TYPE_REAL, pBuffer := ADR(sAux), dwBufferSize := udiAuxBufferSize);
// sAux := TO_STRING(rZmm);
STU.StrConcatA(pstTo := ADR(sZYZ), pstFrom := ADR(sAux), iBufferSize := iBufferSize);

STU.StrConcatA(pstTo := ADR(sZYZ), pstFrom := ADR(';'), iBufferSize := iBufferSize);

sAux := ''; //roll
STU.StuSprintf(pstFormat := ADR('%3.1f'), pVarAdr := ADR(rA), udiVarType := __SYSTEM.TYPE_CLASS.TYPE_REAL, pBuffer := ADR(sAux), dwBufferSize := udiAuxBufferSize);
// sAux := TO_STRING(rRoll);
STU.StrConcatA(pstTo := ADR(sZYZ), pstFrom := ADR(sAux), iBufferSize := iBufferSize);

STU.StrConcatA(pstTo := ADR(sZYZ), pstFrom := ADR(';'), iBufferSize := iBufferSize);

sAux := ''; //pitch
STU.StuSprintf(pstFormat := ADR('%3.1f'), pVarAdr := ADR(rB), udiVarType := __SYSTEM.TYPE_CLASS.TYPE_REAL, pBuffer := ADR(sAux), dwBufferSize := udiAuxBufferSize);
// sAux := TO_STRING(rPitch);
STU.StrConcatA(pstTo := ADR(sZYZ), pstFrom := ADR(sAux), iBufferSize := iBufferSize);

STU.StrConcatA(pstTo := ADR(sZYZ), pstFrom := ADR(';'), iBufferSize := iBufferSize);

sAux := ''; //yaw
STU.StuSprintf(pstFormat := ADR('%3.1f'), pVarAdr := ADR(rC), udiVarType := __SYSTEM.TYPE_CLASS.TYPE_REAL, pBuffer := ADR(sAux), dwBufferSize := udiAuxBufferSize);
// sAux := TO_STRING(rYaw);
STU.StrConcatA(pstTo := ADR(sZYZ), pstFrom := ADR(sAux), iBufferSize := iBufferSize);
                      
END_ACTION

ACTION ACT_Quaternions:
                        // QUATERNION
iBufferSize := TO_INT(XSIZEOF(sQuaternion));
udiAuxBufferSize := TO_UDINT(XSIZEOF(sAux));
sQuaternion := '';


sAux := ''; //X
STU.StuSprintf(pstFormat := ADR('%1.3f'), pVarAdr := ADR(rXMeters), udiVarType := __SYSTEM.TYPE_CLASS.TYPE_REAL, pBuffer := ADR(sAux), dwBufferSize := udiAuxBufferSize); 
// sAux := TO_STRING(rXMeters);
STU.StrConcatA(pstTo := ADR(sQuaternion), pstFrom := ADR(sAux), iBufferSize := iBufferSize);

STU.StrConcatA(pstTo := ADR(sQuaternion), pstFrom := ADR(';'), iBufferSize := iBufferSize);

sAux := ''; //Y
STU.StuSprintf(pstFormat := ADR('%1.3f'), pVarAdr := ADR(rYMeters), udiVarType := __SYSTEM.TYPE_CLASS.TYPE_REAL, pBuffer := ADR(sAux), dwBufferSize := udiAuxBufferSize); 
// sAux := TO_STRING(rYMeters);
STU.StrConcatA(pstTo := ADR(sQuaternion), pstFrom := ADR(sAux), iBufferSize := iBufferSize);

STU.StrConcatA(pstTo := ADR(sQuaternion), pstFrom := ADR(';'), iBufferSize := iBufferSize);

sAux := ''; //Z
STU.StuSprintf(pstFormat := ADR('%1.3f'), pVarAdr := ADR(rZMeters), udiVarType := __SYSTEM.TYPE_CLASS.TYPE_REAL, pBuffer := ADR(sAux), dwBufferSize := udiAuxBufferSize);
// sAux := TO_STRING(rZMeters);
STU.StrConcatA(pstTo := ADR(sQuaternion), pstFrom := ADR(sAux), iBufferSize := iBufferSize);

STU.StrConcatA(pstTo := ADR(sQuaternion), pstFrom := ADR(';'), iBufferSize := iBufferSize);

sAux := ''; //qx
STU.StuSprintf(pstFormat := ADR('%1.3f'), pVarAdr := ADR(rQX), udiVarType := __SYSTEM.TYPE_CLASS.TYPE_REAL, pBuffer := ADR(sAux), dwBufferSize := udiAuxBufferSize);
// sAux := TO_STRING(rQX);
STU.StrConcatA(pstTo := ADR(sQuaternion), pstFrom := ADR(sAux), iBufferSize := iBufferSize);

STU.StrConcatA(pstTo := ADR(sQuaternion), pstFrom := ADR(';'), iBufferSize := iBufferSize);

sAux := ''; //qy
STU.StuSprintf(pstFormat := ADR('%1.3f'), pVarAdr := ADR(rQY), udiVarType := __SYSTEM.TYPE_CLASS.TYPE_REAL, pBuffer := ADR(sAux), dwBufferSize := udiAuxBufferSize);
// sAux := TO_STRING(rQY);
STU.StrConcatA(pstTo := ADR(sQuaternion), pstFrom := ADR(sAux), iBufferSize := iBufferSize);

STU.StrConcatA(pstTo := ADR(sQuaternion), pstFrom := ADR(';'), iBufferSize := iBufferSize);

sAux := ''; //qz
STU.StuSprintf(pstFormat := ADR('%1.3f'), pVarAdr := ADR(rQZ), udiVarType := __SYSTEM.TYPE_CLASS.TYPE_REAL, pBuffer := ADR(sAux), dwBufferSize := udiAuxBufferSize);
// sAux := TO_STRING(rQZ);
STU.StrConcatA(pstTo := ADR(sQuaternion), pstFrom := ADR(sAux), iBufferSize := iBufferSize);

STU.StrConcatA(pstTo := ADR(sQuaternion), pstFrom := ADR(';'), iBufferSize := iBufferSize);

sAux := ''; //qw
STU.StuSprintf(pstFormat := ADR('%1.3f'), pVarAdr := ADR(rQW), udiVarType := __SYSTEM.TYPE_CLASS.TYPE_REAL, pBuffer := ADR(sAux), dwBufferSize := udiAuxBufferSize);
// sAux := TO_STRING(rQW);
STU.StrConcatA(pstTo := ADR(sQuaternion), pstFrom := ADR(sAux), iBufferSize := iBufferSize);
                      
END_ACTION

ACTION ACT_JointsInRadians:
                        IF NOT xINVIS_JointsResults THEN
	IF xConvertToJointRadians THEN
		FOR iIndJoints := 0 TO 5 DO
			arJointsInRadians[iIndJoints] := arJointsInDegrees[iIndJoints] * TO_REAL(SMC_FACTOR_DEG_TO_RAD);
		END_FOR
	END_IF
	
	(*----------------------------------------------*)
	// Radians
	iBufferSize := TO_INT(XSIZEOF(sJointsInRadians));
	udiAuxBufferSize := TO_UDINT(XSIZEOF(sAux));
	sJointsInRadians := '';
	
	sAux := ''; // j1
// 	sAux := TO_STRING(arJointsInRadians[0]);
	STU.StuSprintf(pstFormat := ADR('%3.3f'), pVarAdr := ADR(arJointsInRadians[0]), udiVarType := __SYSTEM.TYPE_CLASS.TYPE_REAL, pBuffer := ADR(sAux), dwBufferSize := udiAuxBufferSize);
	STU.StrConcatA(pstTo := ADR(sJointsInRadians), pstFrom := ADR(sAux), iBufferSize := iBufferSize);
	
	STU.StrConcatA(pstTo := ADR(sJointsInRadians), pstFrom := ADR(';'), iBufferSize := iBufferSize);
	
	sAux := ''; // j2
// 	sAux := TO_STRING(arJointsInRadians[1]);
	STU.StuSprintf(pstFormat := ADR('%3.3f'), pVarAdr := ADR(arJointsInRadians[1]), udiVarType := __SYSTEM.TYPE_CLASS.TYPE_REAL, pBuffer := ADR(sAux), dwBufferSize := udiAuxBufferSize);
	STU.StrConcatA(pstTo := ADR(sJointsInRadians), pstFrom := ADR(sAux), iBufferSize := iBufferSize);
	
	STU.StrConcatA(pstTo := ADR(sJointsInRadians), pstFrom := ADR(';'), iBufferSize := iBufferSize);
	
	sAux := ''; //j3
// 	sAux := TO_STRING(arJointsInRadians[2]);
	STU.StuSprintf(pstFormat := ADR('%3.3f'), pVarAdr := ADR(arJointsInRadians[2]), udiVarType := __SYSTEM.TYPE_CLASS.TYPE_REAL, pBuffer := ADR(sAux), dwBufferSize := udiAuxBufferSize);
	STU.StrConcatA(pstTo := ADR(sJointsInRadians), pstFrom := ADR(sAux), iBufferSize := iBufferSize);
	
	STU.StrConcatA(pstTo := ADR(sJointsInRadians), pstFrom := ADR(';'), iBufferSize := iBufferSize);
	
	sAux := ''; //j4
// 	sAux := TO_STRING(arJointsInRadians[3]);
	STU.StuSprintf(pstFormat := ADR('%3.3f'), pVarAdr := ADR(arJointsInRadians[3]), udiVarType := __SYSTEM.TYPE_CLASS.TYPE_REAL, pBuffer := ADR(sAux), dwBufferSize := udiAuxBufferSize);
	STU.StrConcatA(pstTo := ADR(sJointsInRadians), pstFrom := ADR(sAux), iBufferSize := iBufferSize);
	
	STU.StrConcatA(pstTo := ADR(sJointsInRadians), pstFrom := ADR(';'), iBufferSize := iBufferSize);
	
	sAux := ''; //j5
// 	sAux := TO_STRING(arJointsInRadians[4]);
	STU.StuSprintf(pstFormat := ADR('%3.3f'), pVarAdr := ADR(arJointsInRadians[4]), udiVarType := __SYSTEM.TYPE_CLASS.TYPE_REAL, pBuffer := ADR(sAux), dwBufferSize := udiAuxBufferSize);
	STU.StrConcatA(pstTo := ADR(sJointsInRadians), pstFrom := ADR(sAux), iBufferSize := iBufferSize);
	
	STU.StrConcatA(pstTo := ADR(sJointsInRadians), pstFrom := ADR(';'), iBufferSize := iBufferSize);
	
	sAux := ''; //j6
// 	sAux := TO_STRING(arJointsInRadians[5]);
	STU.StuSprintf(pstFormat := ADR('%3.3f'), pVarAdr := ADR(arJointsInRadians[5]), udiVarType := __SYSTEM.TYPE_CLASS.TYPE_REAL, pBuffer := ADR(sAux), dwBufferSize := udiAuxBufferSize);
	STU.StrConcatA(pstTo := ADR(sJointsInRadians), pstFrom := ADR(sAux), iBufferSize := iBufferSize);
ELSE
	sJointsInRadians := '';
END_IF
                      
END_ACTION

ACTION ACT_JointsInDegrees:
                        IF NOT xINVIS_JointsResults THEN
	IF xConvertToJointDegrees THEN
		FOR iIndJoints := 0 TO 5 DO
			arJointsInDegrees[iIndJoints] := arJointsInRadians[iIndJoints] * TO_REAL(SMC_FACTOR_RAD_TO_DEG);
		END_FOR
	END_IF
	
	(*----------------------------------------------*)
	// Degrees
	iBufferSize := TO_INT(XSIZEOF(sJointsInDegrees));
	udiAuxBufferSize := TO_UDINT(XSIZEOF(sAux));
	

	sJointsInDegrees := '';

	sAux := ''; // j1
// 	sAux := TO_STRING(arJointsInDegrees[0]);
	STU.StuSprintf(pstFormat := ADR('%3.1f'), pVarAdr := ADR(arJointsInDegrees[0]), udiVarType := __SYSTEM.TYPE_CLASS.TYPE_REAL, pBuffer := ADR(sAux), dwBufferSize := udiAuxBufferSize); 
	STU.StrConcatA(pstTo := ADR(sJointsInDegrees), pstFrom := ADR(sAux), iBufferSize := iBufferSize);
	
	STU.StrConcatA(pstTo := ADR(sJointsInDegrees), pstFrom := ADR(';'), iBufferSize := iBufferSize);
	
	sAux := ''; // j2
// 	sAux := TO_STRING(arJointsInDegrees[1]);
	STU.StuSprintf(pstFormat := ADR('%3.1f'), pVarAdr := ADR(arJointsInDegrees[1]), udiVarType := __SYSTEM.TYPE_CLASS.TYPE_REAL, pBuffer := ADR(sAux), dwBufferSize := udiAuxBufferSize); 
	STU.StrConcatA(pstTo := ADR(sJointsInDegrees), pstFrom := ADR(sAux), iBufferSize := iBufferSize);
	
	STU.StrConcatA(pstTo := ADR(sJointsInDegrees), pstFrom := ADR(';'), iBufferSize := iBufferSize);
	
	sAux := ''; //j3
// 	sAux := TO_STRING(arJointsInDegrees[2]);
	STU.StuSprintf(pstFormat := ADR('%3.1f'), pVarAdr := ADR(arJointsInDegrees[2]), udiVarType := __SYSTEM.TYPE_CLASS.TYPE_REAL, pBuffer := ADR(sAux), dwBufferSize := udiAuxBufferSize); 
	STU.StrConcatA(pstTo := ADR(sJointsInDegrees), pstFrom := ADR(sAux), iBufferSize := iBufferSize);
	
	STU.StrConcatA(pstTo := ADR(sJointsInDegrees), pstFrom := ADR(';'), iBufferSize := iBufferSize);
	
	sAux := ''; //j4
// 	sAux := TO_STRING(arJointsInDegrees[3]);
	STU.StuSprintf(pstFormat := ADR('%3.1f'), pVarAdr := ADR(arJointsInDegrees[3]), udiVarType := __SYSTEM.TYPE_CLASS.TYPE_REAL, pBuffer := ADR(sAux), dwBufferSize := udiAuxBufferSize); 
	STU.StrConcatA(pstTo := ADR(sJointsInDegrees), pstFrom := ADR(sAux), iBufferSize := iBufferSize);
	
	STU.StrConcatA(pstTo := ADR(sJointsInDegrees), pstFrom := ADR(';'), iBufferSize := iBufferSize);
	
	sAux := ''; //j5
// 	sAux := TO_STRING(arJointsInDegrees[4]);
	STU.StuSprintf(pstFormat := ADR('%3.1f'), pVarAdr := ADR(arJointsInDegrees[4]), udiVarType := __SYSTEM.TYPE_CLASS.TYPE_REAL, pBuffer := ADR(sAux), dwBufferSize := udiAuxBufferSize); 
	STU.StrConcatA(pstTo := ADR(sJointsInDegrees), pstFrom := ADR(sAux), iBufferSize := iBufferSize);
	
	STU.StrConcatA(pstTo := ADR(sJointsInDegrees), pstFrom := ADR(';'), iBufferSize := iBufferSize);
	
	sAux := ''; //j6
// 	sAux := TO_STRING(arJointsInDegrees[5]);
	STU.StuSprintf(pstFormat := ADR('%3.1f'), pVarAdr := ADR(arJointsInDegrees[5]), udiVarType := __SYSTEM.TYPE_CLASS.TYPE_REAL, pBuffer := ADR(sAux), dwBufferSize := udiAuxBufferSize); 
	STU.StrConcatA(pstTo := ADR(sJointsInDegrees), pstFrom := ADR(sAux), iBufferSize := iBufferSize);
ELSE
	sJointsInDegrees := '';
END_IF

                      
END_ACTION

ACTION ACT_CartConvToMatrix:
                        xIgnoreCart := FALSE;
IF xConvertFromZYZ THEN
	xComputeRotMat := SM3M.SMC_Matrix3_FromZYZ_deg(
		mR := mR,
		dA_deg := arValues[3],
		dB_deg := arValues[4],
		dC_deg := arValues[5]
	);
ELSIF xConvertFromRPY THEN
	xComputeRotMat := SM3M.SMC_Matrix3_FromRollPitchYaw_deg(
		mR := mR,
		dRoll := arValues[3],
		dPitch := arValues[4],
		dYaw := arValues[5]
	);
ELSIF xConvertFromQuat THEN
	quat.dR := arValues[6];
	quat.dI := arValues[3];
	quat.dJ := arValues[4];
	quat.dK := arValues[5];
	SM3M.SMC_Quat1_To_RotMatrix(
		m := mR,
		q := quat
	);
ELSE
	xIgnoreCart := TRUE;
	sZYZ := '';
	sRPY := '';
	sQuaternion := '';
END_IF

IF NOT xIgnoreCart THEN
	
	xIsRot := SM3M.SMC_Matrix3_IsRotation(mR := mR, dEpsRel := 0.001);
	(*-----------------------------*)
	// quaternion conversion from matrix
	SM3M.SMC_Quat1_From_RotMatrix(
		m := mR,
		q := q
	);
	rQW := TO_REAL(q.dR);
	rQX := TO_REAL(q.dI);
	rQY := TO_REAL(q.dJ);
	rQZ := TO_REAL(q.dK);
	(*-----------------------------*)
	// RPY conversion from matrix
	xToRPY := SM3M.SMC_Matrix3_ToRollPitchYaw_deg(
		mR := mR,
		dRoll => lrRoll,
		dPitch => lrPitch,
		dYaw => lrYaw
	);
	rRoll := TO_REAL(lrRoll);
	rPitch := TO_REAL(lrPitch);
	rYaw := TO_REAL(lrYaw);
	(*-----------------------------*)
	// ZYZ conversion from matrix
	xToRPY := SM3M.SMC_Matrix3_ToZYZ_deg(
		mR := mR,
		dA_deg => lrA,
		dB_deg => lrB,
		dC_deg => lrC
	);
	rA := TO_REAL(lrA);
	rB := TO_REAL(lrB);
	rC := TO_REAL(lrC);
	(*-----------------------------*)
	IF xConvertFromZYZ OR xConvertFromRPY THEN
		// mm
		rXmm := arValues[0];
		rYmm := arValues[1];
		rZmm := arValues[2];
		
		// m
		rXMeters := arValues[0]/1000.0;
		rYMeters := arValues[1]/1000.0;
		rZMeters := arValues[2]/1000.0;
	ELSIF xConvertFromQuat THEN
		// mm
		rXmm := arValues[0]*1000.0;
		rYmm := arValues[1]*1000.0;
		rZmm := arValues[2]*1000.0;
		
		// m
		rXMeters := arValues[0];
		rYMeters := arValues[1];
		rZMeters := arValues[2];
	END_IF
	
	ACT_Quaternions();
	ACT_RPY();
	ACT_ZYZ();
END_IF

                      
END_ACTION
END_PROGRAM

PROGRAM prg_Hmi_RobotControl
  VAR
    sDescriptionBar : STRING(255);
    sStatusBar : STRING(255);
    sjAux : STRING;  (* - *)
    sStringJointPos : STRING;
    scAux : STRING;  (* - *)
    sStringCartPos : STRING;
    sQuaternion : STRING(255);
    lrRoll : LREAL;
    lrPitch : LREAL;
    lrYaw : LREAL;
    xToRPY : BOOL;
    rRoll : REAL;
    rPitch : REAL;
    rYaw : REAL;
    rXmm : REAL;
    rYmm : REAL;
    rZmm : REAL;
    sRPY : STRING(255);
    xIsRot : BOOL;
    arJointsInRadians : ARRAY[0..5] OF REAL;
    udiBufferSize : UDINT;
    sJointRadFormatting : STRING := '%1.3f';
    eAdapterError : IoDrvEtherNetIP.DED.ERROR;
    xDiagnosisInfoAvailable : BOOL;
    eAdapterState : IoDrvEtherNetIP.DEVICE_STATE;
    Set_IP : BOOL;
    ipDosan : ARRAY[0..3] OF BYTE;
    deinfo : IoDrvEtherNetIP.DEVICE_INFO;
    errorDE : IoDrvEtherNetIP.DED.ERROR;
    a_ipDoosan : ARRAY[0..3] OF ARRAY[0..3] OF STRING := [['192', '168', '110', '70'], 3([4('')])];
    iIndexIP : INT := 1;  (* -Default impostato sul Doosan *)
    rXMeters : REAL;
    rYMeters : REAL;
    rZMeters : REAL;
    rQW : REAL;
    rQX : REAL;
    rQY : REAL;
    rQZ : REAL;
    mR : SM3M.SMC_Matrix3;
    xComputeRotMat : BOOL;
    q : SM3M.SMC_Quat;
    sAux : STRING(255);
    iBufferSize : INT;
    sJointsInRadians : STRING(255);
  END_VAR

                    IF Set_IP THEN
	Set_IP:=FALSE;		
	ipDosan[0]:=TO_BYTE(a_ipDoosan[0][0]);
	ipDosan[1]:=TO_BYTE(a_ipDoosan[0][1]);
	ipDosan[2]:=TO_BYTE(a_ipDoosan[0][2]);
	ipDosan[3]:=TO_BYTE(a_ipDoosan[0][3]);
	DoosanRobot_EIP_Adapter_Monitoring_GPR.IPAddress:=ipDosan;
END_IF
errorDE:=DoosanRobot_EIP_Adapter_Monitoring_GPR.GetDeviceInfo(deiInfo:=deinfo);
eAdapterState := DoosanRobot_EIP_Adapter_Monitoring_GPR.GetDeviceState(eError => eAdapterError, xDiagnosisInfoAvailable => xDiagnosisInfoAvailable);

ACT_ConcatCartPosString();
ACT_ConcatJointPosString();

ACT_Quaternions();

ACT_JointsInRadians();











                  

ACTION ACT_ConcatJointPosString:
                        // sjAux:=TO_STRING(IO_Variables.EtherNet_IP.Joints.j1);
STU.StuSprintf(pstFormat := ADR('%3.1f'), pVarAdr := ADR(IO_Variables.g_Doosan_EIP.Joints.j1), udiVarType := __SYSTEM.TYPE_CLASS.TYPE_REAL, pBuffer := ADR(sjAux), dwBufferSize := udiBufferSize); 
sStringJointPos:=CONCAT(sjAux,';');

// sjAux:=TO_STRING(IO_Variables.EtherNet_IP.Joints.j2);
STU.StuSprintf(pstFormat := ADR('%3.1f'), pVarAdr := ADR(IO_Variables.g_Doosan_EIP.Joints.j2), udiVarType := __SYSTEM.TYPE_CLASS.TYPE_REAL, pBuffer := ADR(sjAux), dwBufferSize := udiBufferSize); 
sStringJointPos:=CONCAT(sStringJointPos,sjAux);

sjAux:=';';
sStringJointPos:=CONCAT(sStringJointPos,sjAux);

// sjAux:=TO_STRING(IO_Variables.EtherNet_IP.Joints.j3);
STU.StuSprintf(pstFormat := ADR('%3.1f'), pVarAdr := ADR(IO_Variables.g_Doosan_EIP.Joints.j3), udiVarType := __SYSTEM.TYPE_CLASS.TYPE_REAL, pBuffer := ADR(sjAux), dwBufferSize := udiBufferSize); 
sStringJointPos:=CONCAT(sStringJointPos,sjAux);

sjAux:=';';
sStringJointPos:=CONCAT(sStringJointPos,sjAux);

// sjAux:=TO_STRING(IO_Variables.EtherNet_IP.Joints.j4);
STU.StuSprintf(pstFormat := ADR('%3.1f'), pVarAdr := ADR(IO_Variables.g_Doosan_EIP.Joints.j4), udiVarType := __SYSTEM.TYPE_CLASS.TYPE_REAL, pBuffer := ADR(sjAux), dwBufferSize := udiBufferSize); 
sStringJointPos:=CONCAT(sStringJointPos,sjAux);

sjAux:=';';
sStringJointPos:=CONCAT(sStringJointPos,sjAux);

// sjAux:=TO_STRING(IO_Variables.EtherNet_IP.Joints.j5);
STU.StuSprintf(pstFormat := ADR('%3.1f'), pVarAdr := ADR(IO_Variables.g_Doosan_EIP.Joints.j5), udiVarType := __SYSTEM.TYPE_CLASS.TYPE_REAL, pBuffer := ADR(sjAux), dwBufferSize := udiBufferSize); 
sStringJointPos:=CONCAT(sStringJointPos,sjAux);

sjAux:=';';
sStringJointPos:=CONCAT(sStringJointPos,sjAux);

// sjAux:=TO_STRING(IO_Variables.EtherNet_IP.Joints.j6);
STU.StuSprintf(pstFormat := ADR('%3.1f'), pVarAdr := ADR(IO_Variables.g_Doosan_EIP.Joints.j6), udiVarType := __SYSTEM.TYPE_CLASS.TYPE_REAL, pBuffer := ADR(sjAux), dwBufferSize := udiBufferSize); 
sStringJointPos:=CONCAT(sStringJointPos,sjAux);

                      
END_ACTION

ACTION ACT_ConcatCartPosString:
                        // scAux:=TO_STRING(IO_Variables.EtherNet_IP.Cartesian.x);
STU.StuSprintf(pstFormat := ADR('%3.1f'), pVarAdr := ADR(IO_Variables.g_Doosan_EIP.Cartesian.x), udiVarType := __SYSTEM.TYPE_CLASS.TYPE_REAL, pBuffer := ADR(scAux), dwBufferSize := udiBufferSize); 
sStringCartPos:=CONCAT(scAux,';');

// scAux:=TO_STRING(IO_Variables.EtherNet_IP.Cartesian.y);
STU.StuSprintf(pstFormat := ADR('%3.1f'), pVarAdr := ADR(IO_Variables.g_Doosan_EIP.Cartesian.y), udiVarType := __SYSTEM.TYPE_CLASS.TYPE_REAL, pBuffer := ADR(scAux), dwBufferSize := udiBufferSize); 
sStringCartPos:=CONCAT(sStringCartPos,scAux);

scAux:=';';
sStringCartPos:=CONCAT(sStringCartPos,scAux);

// scAux:=TO_STRING(IO_Variables.EtherNet_IP.Cartesian.z);
STU.StuSprintf(pstFormat := ADR('%3.1f'), pVarAdr := ADR(IO_Variables.g_Doosan_EIP.Cartesian.z), udiVarType := __SYSTEM.TYPE_CLASS.TYPE_REAL, pBuffer := ADR(scAux), dwBufferSize := udiBufferSize); 
sStringCartPos:=CONCAT(sStringCartPos,scAux);

scAux:=';';
sStringCartPos:=CONCAT(sStringCartPos,scAux);

// scAux:=TO_STRING(IO_Variables.EtherNet_IP.Cartesian.A);
STU.StuSprintf(pstFormat := ADR('%3.1f'), pVarAdr := ADR(IO_Variables.g_Doosan_EIP.Cartesian.A), udiVarType := __SYSTEM.TYPE_CLASS.TYPE_REAL, pBuffer := ADR(scAux), dwBufferSize := udiBufferSize); 
sStringCartPos:=CONCAT(sStringCartPos,scAux);

scAux:=';';
sStringCartPos:=CONCAT(sStringCartPos,scAux);

// scAux:=TO_STRING(IO_Variables.EtherNet_IP.Cartesian.B);
STU.StuSprintf(pstFormat := ADR('%3.1f'), pVarAdr := ADR(IO_Variables.g_Doosan_EIP.Cartesian.B), udiVarType := __SYSTEM.TYPE_CLASS.TYPE_REAL, pBuffer := ADR(scAux), dwBufferSize := udiBufferSize); 
sStringCartPos:=CONCAT(sStringCartPos,scAux);

scAux:=';';
sStringCartPos:=CONCAT(sStringCartPos,scAux);

// scAux:=TO_STRING(IO_Variables.EtherNet_IP.Cartesian.C);
STU.StuSprintf(pstFormat := ADR('%3.1f'), pVarAdr := ADR(IO_Variables.g_Doosan_EIP.Cartesian.C), udiVarType := __SYSTEM.TYPE_CLASS.TYPE_REAL, pBuffer := ADR(scAux), dwBufferSize := udiBufferSize); 
sStringCartPos:=CONCAT(sStringCartPos,scAux);

                      
END_ACTION

ACTION ACT_Quaternions:
                        xComputeRotMat := SM3M.SMC_Matrix3_FromZYZ_deg(
	mR := mR,
	dA_deg := IO_Variables.g_Doosan_EIP.Cartesian.A,
	dB_deg := IO_Variables.g_Doosan_EIP.Cartesian.B,
	dC_deg := IO_Variables.g_Doosan_EIP.Cartesian.C
);

// xComputeRotMat := SM3M.SMC_Matrix3_FromRollPitchYaw_deg(
// 	mR := mR,
// 	dRoll := IO_Variables.EtherNet_IP.Cartesian.A,
// 	dPitch := IO_Variables.EtherNet_IP.Cartesian.B,
// 	dYaw := IO_Variables.EtherNet_IP.Cartesian.C
// );

xIsRot := SM3M.SMC_Matrix3_IsRotation(mR := mR, dEpsRel := 0.001);

SM3M.SMC_Quat1_From_RotMatrix(
	m := mR,
	q := q
);

xToRPY := SM3M.SMC_Matrix3_ToRollPitchYaw_deg(
	mR := mR,
	dRoll => lrRoll,
	dPitch => lrPitch,
	dYaw => lrYaw
);

/// quaternions
iBufferSize := TO_INT(XSIZEOF(sQuaternion));
sQuaternion := '';

// ROUND

rXmm := TO_REAL(IO_Variables.g_Doosan_EIP.Cartesian.x);
rYmm := TO_REAL(IO_Variables.g_Doosan_EIP.Cartesian.y);
rZmm := TO_REAL(IO_Variables.g_Doosan_EIP.Cartesian.z);

rXMeters := rXmm / 1000.0;
rYMeters := rYmm / 1000.0;
rZMeters := rZmm / 1000.0;

// rQW := TO_REAL(TO_INT(q.dR * 1E6)) / 1E6;
// rQX := TO_REAL(TO_INT(q.dI * 1E6)) / 1E6;
// rQY := TO_REAL(TO_INT(q.dJ * 1E6)) / 1E6;
// rQZ := TO_REAL(TO_INT(q.dK * 1E6)) / 1E6;
rQW := TO_REAL(q.dR);
rQX := TO_REAL(q.dI);
rQY := TO_REAL(q.dJ);
rQZ := TO_REAL(q.dK);

rRoll := TO_REAL(lrRoll);
rPitch := TO_REAL(lrPitch);
rYaw := TO_REAL(lrYaw);

// QUATERNION
sAux := ''; //X
STU.StuSprintf(pstFormat := ADR('%1.3f'), pVarAdr := ADR(rXMeters), udiVarType := __SYSTEM.TYPE_CLASS.TYPE_REAL, pBuffer := ADR(sAux), dwBufferSize := udiBufferSize); 
// sAux := TO_STRING(rXMeters);
STU.StrConcatA(pstTo := ADR(sQuaternion), pstFrom := ADR(sAux), iBufferSize := iBufferSize);

STU.StrConcatA(pstTo := ADR(sQuaternion), pstFrom := ADR(';'), iBufferSize := iBufferSize);

sAux := ''; //Y
STU.StuSprintf(pstFormat := ADR('%1.3f'), pVarAdr := ADR(rYMeters), udiVarType := __SYSTEM.TYPE_CLASS.TYPE_REAL, pBuffer := ADR(sAux), dwBufferSize := udiBufferSize); 
// sAux := TO_STRING(rYMeters);
STU.StrConcatA(pstTo := ADR(sQuaternion), pstFrom := ADR(sAux), iBufferSize := iBufferSize);

STU.StrConcatA(pstTo := ADR(sQuaternion), pstFrom := ADR(';'), iBufferSize := iBufferSize);

sAux := ''; //Z
STU.StuSprintf(pstFormat := ADR('%1.3f'), pVarAdr := ADR(rZMeters), udiVarType := __SYSTEM.TYPE_CLASS.TYPE_REAL, pBuffer := ADR(sAux), dwBufferSize := udiBufferSize);
// sAux := TO_STRING(rZMeters);
STU.StrConcatA(pstTo := ADR(sQuaternion), pstFrom := ADR(sAux), iBufferSize := iBufferSize);

STU.StrConcatA(pstTo := ADR(sQuaternion), pstFrom := ADR(';'), iBufferSize := iBufferSize);

sAux := ''; //qx
STU.StuSprintf(pstFormat := ADR('%1.3f'), pVarAdr := ADR(rQX), udiVarType := __SYSTEM.TYPE_CLASS.TYPE_REAL, pBuffer := ADR(sAux), dwBufferSize := udiBufferSize);
// sAux := TO_STRING(rQX);
STU.StrConcatA(pstTo := ADR(sQuaternion), pstFrom := ADR(sAux), iBufferSize := iBufferSize);

STU.StrConcatA(pstTo := ADR(sQuaternion), pstFrom := ADR(';'), iBufferSize := iBufferSize);

sAux := ''; //qy
STU.StuSprintf(pstFormat := ADR('%1.3f'), pVarAdr := ADR(rQY), udiVarType := __SYSTEM.TYPE_CLASS.TYPE_REAL, pBuffer := ADR(sAux), dwBufferSize := udiBufferSize);
// sAux := TO_STRING(rQY);
STU.StrConcatA(pstTo := ADR(sQuaternion), pstFrom := ADR(sAux), iBufferSize := iBufferSize);

STU.StrConcatA(pstTo := ADR(sQuaternion), pstFrom := ADR(';'), iBufferSize := iBufferSize);

sAux := ''; //qz
STU.StuSprintf(pstFormat := ADR('%1.3f'), pVarAdr := ADR(rQZ), udiVarType := __SYSTEM.TYPE_CLASS.TYPE_REAL, pBuffer := ADR(sAux), dwBufferSize := udiBufferSize);
// sAux := TO_STRING(rQZ);
STU.StrConcatA(pstTo := ADR(sQuaternion), pstFrom := ADR(sAux), iBufferSize := iBufferSize);

STU.StrConcatA(pstTo := ADR(sQuaternion), pstFrom := ADR(';'), iBufferSize := iBufferSize);

sAux := ''; //qw
STU.StuSprintf(pstFormat := ADR('%1.3f'), pVarAdr := ADR(rQW), udiVarType := __SYSTEM.TYPE_CLASS.TYPE_REAL, pBuffer := ADR(sAux), dwBufferSize := udiBufferSize);
// sAux := TO_STRING(rQW);
STU.StrConcatA(pstTo := ADR(sQuaternion), pstFrom := ADR(sAux), iBufferSize := iBufferSize);

(*----------------------------------------------*)
// RPY
iBufferSize := TO_INT(XSIZEOF(sRPY));
sRPY := '';

sAux := ''; //X
STU.StuSprintf(pstFormat := ADR('%5.1f'), pVarAdr := ADR(rXmm), udiVarType := __SYSTEM.TYPE_CLASS.TYPE_REAL, pBuffer := ADR(sAux), dwBufferSize := udiBufferSize);
// sAux := TO_STRING(rXmm);
STU.StrConcatA(pstTo := ADR(sRPY), pstFrom := ADR(sAux), iBufferSize := iBufferSize);

STU.StrConcatA(pstTo := ADR(sRPY), pstFrom := ADR(';'), iBufferSize := iBufferSize);

sAux := ''; //Y
STU.StuSprintf(pstFormat := ADR('%5.1f'), pVarAdr := ADR(rYmm), udiVarType := __SYSTEM.TYPE_CLASS.TYPE_REAL, pBuffer := ADR(sAux), dwBufferSize := udiBufferSize);
// sAux := TO_STRING(rYmm);
STU.StrConcatA(pstTo := ADR(sRPY), pstFrom := ADR(sAux), iBufferSize := iBufferSize);

STU.StrConcatA(pstTo := ADR(sRPY), pstFrom := ADR(';'), iBufferSize := iBufferSize);

sAux := ''; //Z
STU.StuSprintf(pstFormat := ADR('%5.1f'), pVarAdr := ADR(rZmm), udiVarType := __SYSTEM.TYPE_CLASS.TYPE_REAL, pBuffer := ADR(sAux), dwBufferSize := udiBufferSize);
// sAux := TO_STRING(rZmm);
STU.StrConcatA(pstTo := ADR(sRPY), pstFrom := ADR(sAux), iBufferSize := iBufferSize);

STU.StrConcatA(pstTo := ADR(sRPY), pstFrom := ADR(';'), iBufferSize := iBufferSize);

sAux := ''; //roll
STU.StuSprintf(pstFormat := ADR('%3.1f'), pVarAdr := ADR(rRoll), udiVarType := __SYSTEM.TYPE_CLASS.TYPE_REAL, pBuffer := ADR(sAux), dwBufferSize := udiBufferSize);
// sAux := TO_STRING(rRoll);
STU.StrConcatA(pstTo := ADR(sRPY), pstFrom := ADR(sAux), iBufferSize := iBufferSize);

STU.StrConcatA(pstTo := ADR(sRPY), pstFrom := ADR(';'), iBufferSize := iBufferSize);

sAux := ''; //pitch
STU.StuSprintf(pstFormat := ADR('%3.1f'), pVarAdr := ADR(rPitch), udiVarType := __SYSTEM.TYPE_CLASS.TYPE_REAL, pBuffer := ADR(sAux), dwBufferSize := udiBufferSize);
// sAux := TO_STRING(rPitch);
STU.StrConcatA(pstTo := ADR(sRPY), pstFrom := ADR(sAux), iBufferSize := iBufferSize);

STU.StrConcatA(pstTo := ADR(sRPY), pstFrom := ADR(';'), iBufferSize := iBufferSize);

sAux := ''; //yaw
STU.StuSprintf(pstFormat := ADR('%3.1f'), pVarAdr := ADR(rYaw), udiVarType := __SYSTEM.TYPE_CLASS.TYPE_REAL, pBuffer := ADR(sAux), dwBufferSize := udiBufferSize);
// sAux := TO_STRING(rYaw);
STU.StrConcatA(pstTo := ADR(sRPY), pstFrom := ADR(sAux), iBufferSize := iBufferSize);

                      
END_ACTION

ACTION ACT_JointsInRadians:
                        arJointsInRadians[0] := IO_Variables.g_Doosan_EIP.Joints.j1 * TO_REAL(SMC_FACTOR_DEG_TO_RAD);
arJointsInRadians[1] := IO_Variables.g_Doosan_EIP.Joints.j2 * TO_REAL(SMC_FACTOR_DEG_TO_RAD);
arJointsInRadians[2] := IO_Variables.g_Doosan_EIP.Joints.j3 * TO_REAL(SMC_FACTOR_DEG_TO_RAD);
arJointsInRadians[3] := IO_Variables.g_Doosan_EIP.Joints.j4 * TO_REAL(SMC_FACTOR_DEG_TO_RAD);
arJointsInRadians[4] := IO_Variables.g_Doosan_EIP.Joints.j5 * TO_REAL(SMC_FACTOR_DEG_TO_RAD);
arJointsInRadians[5] := IO_Variables.g_Doosan_EIP.Joints.j6 * TO_REAL(SMC_FACTOR_DEG_TO_RAD);


(*----------------------------------------------*)
// Radians
iBufferSize := TO_INT(XSIZEOF(sJointsInRadians));
udiBufferSize := TO_UDINT(XSIZEOF(sJointsInRadians));
sJointsInRadians := '';

sAux := ''; // j1
STU.StuSprintf(pstFormat := ADR('%1.3f'), pVarAdr := ADR(arJointsInRadians[0]), udiVarType := __SYSTEM.TYPE_CLASS.TYPE_REAL, pBuffer := ADR(sAux), dwBufferSize := udiBufferSize); 
// sAux := TO_STRING(arJointsInRadians[0]);
STU.StrConcatA(pstTo := ADR(sJointsInRadians), pstFrom := ADR(sAux), iBufferSize := iBufferSize);

STU.StrConcatA(pstTo := ADR(sJointsInRadians), pstFrom := ADR(';'), iBufferSize := iBufferSize);

sAux := ''; // j2
STU.StuSprintf(pstFormat := ADR('%1.3f'), pVarAdr := ADR(arJointsInRadians[1]), udiVarType := __SYSTEM.TYPE_CLASS.TYPE_REAL, pBuffer := ADR(sAux), dwBufferSize := udiBufferSize); 
// sAux := TO_STRING(arJointsInRadians[1]);
STU.StrConcatA(pstTo := ADR(sJointsInRadians), pstFrom := ADR(sAux), iBufferSize := iBufferSize);

STU.StrConcatA(pstTo := ADR(sJointsInRadians), pstFrom := ADR(';'), iBufferSize := iBufferSize);

sAux := ''; //j3
STU.StuSprintf(pstFormat := ADR('%1.3f'), pVarAdr := ADR(arJointsInRadians[2]), udiVarType := __SYSTEM.TYPE_CLASS.TYPE_REAL, pBuffer := ADR(sAux), dwBufferSize := udiBufferSize); 
// sAux := TO_STRING(arJointsInRadians[2]);
STU.StrConcatA(pstTo := ADR(sJointsInRadians), pstFrom := ADR(sAux), iBufferSize := iBufferSize);

STU.StrConcatA(pstTo := ADR(sJointsInRadians), pstFrom := ADR(';'), iBufferSize := iBufferSize);

sAux := ''; //j4
STU.StuSprintf(pstFormat := ADR('%1.3f'), pVarAdr := ADR(arJointsInRadians[3]), udiVarType := __SYSTEM.TYPE_CLASS.TYPE_REAL, pBuffer := ADR(sAux), dwBufferSize := udiBufferSize); 
// sAux := TO_STRING(arJointsInRadians[3]);
STU.StrConcatA(pstTo := ADR(sJointsInRadians), pstFrom := ADR(sAux), iBufferSize := iBufferSize);

STU.StrConcatA(pstTo := ADR(sJointsInRadians), pstFrom := ADR(';'), iBufferSize := iBufferSize);

sAux := ''; //j5
STU.StuSprintf(pstFormat := ADR('%1.3f'), pVarAdr := ADR(arJointsInRadians[4]), udiVarType := __SYSTEM.TYPE_CLASS.TYPE_REAL, pBuffer := ADR(sAux), dwBufferSize := udiBufferSize); 
// sAux := TO_STRING(arJointsInRadians[4]);
STU.StrConcatA(pstTo := ADR(sJointsInRadians), pstFrom := ADR(sAux), iBufferSize := iBufferSize);

STU.StrConcatA(pstTo := ADR(sJointsInRadians), pstFrom := ADR(';'), iBufferSize := iBufferSize);

sAux := ''; //j6
STU.StuSprintf(pstFormat := ADR('%1.3f'), pVarAdr := ADR(arJointsInRadians[5]), udiVarType := __SYSTEM.TYPE_CLASS.TYPE_REAL, pBuffer := ADR(sAux), dwBufferSize := udiBufferSize); 
// sAux := TO_STRING(arJointsInRadians[5]);
STU.StrConcatA(pstTo := ADR(sJointsInRadians), pstFrom := ADR(sAux), iBufferSize := iBufferSize);
                      
END_ACTION
END_PROGRAM

PROGRAM prg_Hmi_PalletConfig
  VAR
    sPalletConfigDescr : STRING;
    xTB_SelectPalletConfig01 : BOOL;
    xDIS_SelectPalletConfig01 : BOOL;
    xTB_SelectPalletConfig02 : BOOL;
    xDIS_SelectPalletConfig02 : BOOL;
    xTB_AirOff : BOOL;
    sDescriptionBar : STRING(255) := 'Stato config pallet:';
    sStatusMessage : STRING(255);
  END_VAR

                    CASE PersVars.g_uiCurrentPalletConfig OF
	GVL_Constants.gc_uiPalletConfigIndex_01:
		sPalletConfigDescr := 'PALL CONFIG 01';
	GVL_Constants.gc_uiPalletConfigIndex_02:
		sPalletConfigDescr := 'PALL CONFIG 02';
	ELSE
		sPalletConfigDescr := 'Unknown pallet config';
END_CASE
(**)
// pallet config selection
xDIS_SelectPalletConfig01 := prgMain.METH_IsPalletConfig01() OR GVL.g_xRUNNING;
IF xTB_SelectPalletConfig01 THEN
	xTB_SelectPalletConfig01 := FALSE;
	prgMain.METH_SetPalletConfig01();
END_IF

xDIS_SelectPalletConfig02 := prgMain.METH_IsPalletConfig02() OR GVL.g_xRUNNING;
IF xTB_SelectPalletConfig02 THEN
	xTB_SelectPalletConfig02 := FALSE;
	prgMain.METH_SetPalletConfig02();
END_IF
(**)
IF xTB_AirOff THEN
	xTB_AirOff := FALSE;
	
END_IF
                  
END_PROGRAM

(* Event handler for mouse events. *)
FUNCTION_BLOCK EventHandler IMPLEMENTS VisuElems.VisuElemBase.IMouseEventHandler
  VAR_INPUT
    mouseMove : REFERENCE TO MouseInfo;
    mouseDown : REFERENCE TO MouseInfo;
    mouseUp : REFERENCE TO MouseInfo;
  END_VAR

                    
                  

(* This method will be called when a mouse button is pressed. RETURN: TRUE - When the handler has handled this event and it should not be handled by someone else FALSE - When the event is not handled by this handler *)
METHOD HandleMouseBtnEvent : BOOL
  VAR_INPUT
    bMouseUpEvent : BOOL;  (* The event type. The value is true if a mouse button was released. *)
    btMouseBtn : BYTE;  (* Information about the button that was pressed or released. At the moment this value is not yet used and will always have the value 0! *)
    ptMouse : VisuElems.CmpVisuHandler.VisuStructPoint;  (* The position where the mouse event was raised. *)
    pClient : POINTER TO VisuElems.VisuStructClientData;  (* A pointer to the client structure were the event occurred. *)
  END_VAR
  VAR
    pDestEvent : POINTER TO MouseInfo;
  END_VAR
                          IF bMouseUpEvent THEN
	pDestEvent := ADR(mouseUp);
ELSE
	pDestEvent := ADR(mouseDown);
END_IF

pDestEvent^.eventCounter := pDestEvent^.eventCounter + 1;
pDestEvent^.iX := ptMouse.iX;
pDestEvent^.iY := ptMouse.iY;

                        
END_METHOD

(* This method will be called when the mouse was moved. RETURN: TRUE - When the handler has handled this event and it should not be handled by someone else FALSE - When the event is not handled by this handler *)
METHOD HandleMouseMoveEvent : BOOL
  VAR_INPUT
    ptMouse : VisuElems.CmpVisuHandler.VisuStructPoint;  (* The position where the mouse was moved to. *)
    pClient : POINTER TO VisuElems.VisuStructClientData;  (* A pointer to the client structure were the event occurred. *)
  END_VAR
                          mouseMove.eventCounter := mouseMove.eventCounter + 1;
mouseMove.iX := ptMouse.iX;
mouseMove.iY := ptMouse.iY;

                        
END_METHOD
END_FUNCTION_BLOCK

(* Helper function block with mouse infos like position, event counter and event type. *)
FUNCTION_BLOCK MouseInfo
  VAR_INPUT
    stType : STRING;
    iX : INT;
    iY : INT;
    eventCounter : INT;
  END_VAR

                    
                  
END_FUNCTION_BLOCK

(* This example show how the mouse event handler is used. *)
PROGRAM PLC_PRG
  VAR
    lastMove : MouseInfo := (stType := 'Move', iX := -1, iY := -1);  (* Helper function block for 'move' events *)
    lastDown : MouseInfo := (stType := 'Down', iX := -1, iY := -1);  (* Helper function block for 'down' events *)
    lastUp : MouseInfo := (stType := 'Up', iX := -1, iY := -1);  (* Helper function block for 'up' events *)
    evHandler : EventHandler;  (* implements VisuElems.VisuElemBase.IMouseEventHandler *)
    bInit : BOOL := TRUE;
  END_VAR

                    // Set up mouse info helper
IF bInit THEN
	bInit := FALSE;	
	evHandler.mouseUp REF= lastUp;
	evHandler.mouseDown REF= lastDown;
	evHandler.mouseMove REF= lastMove;
END_IF

                  
END_PROGRAM

(* This function is called after visu initialization (see Visualization Manager 'Call after visu initialization') *)
FUNCTION VisuInit : BOOL

                    // Set the mouse event handler
VisuElems.VisuElemBase.g_VisuEventManager.SetMouseEventHandler(PLC_PRG.evHandler);

                  
END_FUNCTION

PROGRAM prg_Hmi_ZoneTractor
  VAR
    i : INT;
    iInputWight : INT;
    iInputHeight : INT;
    xApplyDimentions : BOOL;
    a_iMoveX : ARRAY[0..c_iMaxZone] OF INT;
    a_iMoveY : ARRAY[0..c_iMaxZone] OF INT;
    a_iSaveCurrentPosX : ARRAY[0..c_iMaxZone] OF INT;
    a_iSaveCurrentPosY : ARRAY[0..c_iMaxZone] OF INT;
    a_iWight : ARRAY[0..c_iMaxZone] OF INT;  (* - *)
    a_iHeight : ARRAY[0..c_iMaxZone] OF INT;
    a_sPositionRectangle : ARRAY[0..c_iMaxZone] OF STRING(255);  (* - *)
    a_xEnableMove : ARRAY[0..c_iMaxZone] OF BOOL;  (* - *)
    a_xEnableBlocks : ARRAY[0..c_iMaxZone] OF BOOL := [TRUE, 18(FALSE), TRUE, FALSE];  (* - *)
    i_IndexSelection : INT;  (* - *)
    xEnableNewBlock : BOOL;
    zones : ARRAY[0..c_iMaxZone] OF zones_t := [19(()), (a_iMoveX := 25, a_iMoveY := 2, a_iSaveCurrentPosX := 2, a_iSaveCurrentPosY := 2, a_xEnableBlocks := TRUE), ()];  (* - *)
    zones_Empty : ARRAY[0..c_iMaxZone] OF zones_t := [19(()), (a_iMoveX := 25, a_iMoveY := 2, a_iSaveCurrentPosX := 25, a_iSaveCurrentPosY := 2, a_xEnableBlocks := TRUE), ()];
    zones_FirstPattern : ARRAY[0..c_iMaxZone] OF zones_t := [(a_iMoveX := 446, a_iMoveY := 36, a_iSaveCurrentPosX := 446, a_iSaveCurrentPosY := 36, a_iWight := 260, a_iHeight := 370, a_xEnableBlocks := TRUE), (a_iMoveX := 446, a_iMoveY := 354, a_iSaveCurrentPosX := 446, a_iSaveCurrentPosY := 354, a_iWight := 260, a_iHeight := 360, a_xEnableBlocks := TRUE), (a_iMoveX := 656, a_iMoveY := 36, a_iSaveCurrentPosX := 656, a_iSaveCurrentPosY := 36, a_iWight := 400, a_iHeight := 260, a_xEnableBlocks := TRUE), (a_iMoveX := 656, a_iMoveY := 244, a_iSaveCurrentPosX := 656, a_iSaveCurrentPosY := 244, a_iWight := 400, a_iHeight := 260, a_xEnableBlocks := TRUE), (a_iMoveX := 656, a_iMoveY := 454, a_iSaveCurrentPosX := 656, a_iSaveCurrentPosY := 454, a_iWight := 400, a_iHeight := 260, a_xEnableBlocks := TRUE), (a_iMoveX := 1006, a_iMoveY := 36, a_iSaveCurrentPosX := 1006, a_iSaveCurrentPosY := 36, a_iWight := 400, a_iHeight := 260, a_xEnableBlocks := TRUE), (a_iMoveX := 1006, a_iMoveY := 244, a_iSaveCurrentPosX := 1006, a_iSaveCurrentPosY := 244, a_iWight := 400, a_iHeight := 260, a_xEnableBlocks := TRUE), (a_iMoveX := 1006, a_iMoveY := 454, a_iSaveCurrentPosX := 1006, a_iSaveCurrentPosY := 454, a_iWight := 400, a_iHeight := 260, a_xEnableBlocks := TRUE), 11(()), (a_iMoveX := 7, a_iMoveY := -26, a_iSaveCurrentPosX := 7, a_iSaveCurrentPosY := -26, a_iWight := 80, a_iHeight := 60, a_xEnableBlocks := TRUE), ()];
    zones_SecondPattern : ARRAY[0..c_iMaxZone] OF zones_t := [(a_iMoveX := 446, a_iMoveY := 1, a_iSaveCurrentPosX := 446, a_iSaveCurrentPosY := 1, a_iWight := 260, a_iHeight := 400, a_xEnableBlocks := TRUE), (a_iMoveX := 446, a_iMoveY := 351, a_iSaveCurrentPosX := 446, a_iSaveCurrentPosY := 351, a_iWight := 260, a_iHeight := 400, a_xEnableBlocks := TRUE), (a_iMoveX := 656, a_iMoveY := 1, a_iSaveCurrentPosX := 656, a_iSaveCurrentPosY := 1, a_iWight := 260, a_iHeight := 400, a_xEnableBlocks := TRUE), (a_iMoveX := 656, a_iMoveY := 351, a_iSaveCurrentPosX := 656, a_iSaveCurrentPosY := 351, a_iWight := 260, a_iHeight := 400, a_xEnableBlocks := TRUE), (a_iMoveX := 865, a_iMoveY := 1, a_iSaveCurrentPosX := 865, a_iSaveCurrentPosY := 1, a_iWight := 260, a_iHeight := 400, a_xEnableBlocks := TRUE), (a_iMoveX := 865, a_iMoveY := 351, a_iSaveCurrentPosX := 865, a_iSaveCurrentPosY := 351, a_iWight := 260, a_iHeight := 400, a_xEnableBlocks := TRUE), (a_iMoveX := 1075, a_iMoveY := 1, a_iSaveCurrentPosX := 1075, a_iSaveCurrentPosY := 1, a_iWight := 260, a_iHeight := 400, a_xEnableBlocks := TRUE), (a_iMoveX := 1075, a_iMoveY := 351, a_iSaveCurrentPosX := 1075, a_iSaveCurrentPosY := 351, a_iWight := 260, a_iHeight := 400, a_xEnableBlocks := TRUE), 11(()), (a_iMoveX := -54, a_iMoveY := 3, a_iSaveCurrentPosX := -54, a_iSaveCurrentPosY := 3, a_iWight := 130, a_xEnableBlocks := TRUE), ()];
    zones_FirstPattern_backup : ARRAY[0..c_iMaxZone] OF zones_t := [(a_iMoveX := 441, a_iMoveY := 114, a_iSaveCurrentPosX := 441, a_iSaveCurrentPosY := 114, a_iWight := 260, a_iHeight := 400, a_xEnableBlocks := TRUE), (a_iMoveX := 446, a_iMoveY := 514, a_iSaveCurrentPosX := 446, a_iSaveCurrentPosY := 514, a_iWight := 260, a_iHeight := 400, a_xEnableBlocks := TRUE), (a_iMoveX := 706, a_iMoveY := 124, a_iSaveCurrentPosX := 706, a_iSaveCurrentPosY := 124, a_iWight := 400, a_iHeight := 260, a_xEnableBlocks := TRUE), (a_iMoveX := 706, a_iMoveY := 384, a_iSaveCurrentPosX := 706, a_iSaveCurrentPosY := 384, a_iWight := 400, a_iHeight := 260, a_xEnableBlocks := TRUE), (a_iMoveX := 706, a_iMoveY := 644, a_iSaveCurrentPosX := 706, a_iSaveCurrentPosY := 644, a_iWight := 400, a_iHeight := 260, a_xEnableBlocks := TRUE), (a_iMoveX := 1106, a_iMoveY := 124, a_iSaveCurrentPosX := 1106, a_iSaveCurrentPosY := 124, a_iWight := 400, a_iHeight := 260, a_xEnableBlocks := TRUE), (a_iMoveX := 1106, a_iMoveY := 384, a_iSaveCurrentPosX := 1106, a_iSaveCurrentPosY := 384, a_iWight := 400, a_iHeight := 260, a_xEnableBlocks := TRUE), (a_iMoveX := 1106, a_iMoveY := 644, a_iSaveCurrentPosX := 1106, a_iSaveCurrentPosY := 644, a_iWight := 400, a_iHeight := 260, a_xEnableBlocks := TRUE), 11(()), (a_iMoveX := 25, a_iMoveY := 2, a_iSaveCurrentPosX := 25, a_iSaveCurrentPosY := 2, a_xEnableBlocks := TRUE), ()];
    xSave : BOOL;
    xLoad : BOOL;
    x : INT;
    xchargeParams : BOOL;
    iConfSave : INT;
    xReloadTrasportLocalParam : BOOL;
    xReloadFirstPattern : BOOL;
    xReloadSecondPattern : BOOL;
    xChargeEmpty : BOOL;
  END_VAR
  VAR CONSTANT
    c_iMaxZone : INT := 20;
  END_VAR

                    // sPositionRectangle:=Concat('x',Concat(TO_STRING(iMoveX),Concat('$Ny',TO_STRING(iMoveY))));
// iWight:=iInputWight*-1;
// iHeight:=iInputHeight*-1;
// 
// IF xEnableMove THEN
// 	iMoveX:=(PLC_PRG.lastMove.iX-PLC_PRG.lastDown.iX)+iSaveCurrentPosX;
// 	iMoveY:=(PLC_PRG.lastMove.iY-PLC_PRG.lastDown.iY)+iSaveCurrentPosY;
// END_IF
//--------------------------------------------------------------------------------------------------//
FOR i:=0 TO c_iMaxZone DO
	IF xEnableNewBlock AND NOT a_xEnableBlocks[i] THEN
		xEnableNewBlock:=FALSE;
		a_xEnableBlocks[i]:=TRUE;
	END_IF
END_FOR

// a_sPositionRectangle[i_IndexSelection]:=Concat('x',Concat(TO_STRING(a_iMoveX[i_IndexSelection]),Concat('$Ny',TO_STRING(a_iMoveY[i_IndexSelection]))));
IF xApplyDimentions THEN
	xApplyDimentions:=FALSE;
	a_iWight[i_IndexSelection]:=(iInputWight*-1)+100;
	a_iHeight[i_IndexSelection]:=(iInputHeight*-1)+100;
END_IF
IF a_xEnableMove[i_IndexSelection] THEN
	a_iMoveX[i_IndexSelection]:=(PLC_PRG.lastMove.iX-PLC_PRG.lastDown.iX)+a_iSaveCurrentPosX[i_IndexSelection];
	a_iMoveY[i_IndexSelection]:=(PLC_PRG.lastMove.iY-PLC_PRG.lastDown.iY)+a_iSaveCurrentPosY[i_IndexSelection];
	
END_IF
//----------------------------------------------------------------------------------------------------------------------//
IF xchargeParams THEN
	xchargeParams:=FALSE;
	FOR x:=0 TO c_iMaxZone DO
		zones[x].a_sPositionRectangle:=a_sPositionRectangle[x];
		zones[x].a_iWight:=a_iWight[x];
		zones[x].a_iHeight:=a_iHeight[x];
		
			//-
		zones[x].a_iMoveX:=a_iMoveX[x];
		zones[x].a_iMoveY:=a_iMoveY[x];
			//-
		zones[x].a_xEnableBlocks:=a_xEnableBlocks[x];
		zones[x].a_iSaveCurrentPosX:=a_iSaveCurrentPosX[x];
		zones[x].a_iSaveCurrentPosY:=a_iSaveCurrentPosY[x];
	END_FOR
END_IF
IF xReloadTrasportLocalParam THEN
	xReloadTrasportLocalParam:=FALSE;
	FOR x:=0 TO c_iMaxZone DO
		a_sPositionRectangle[x]:=zones[x].a_sPositionRectangle;
		a_iWight[x]:=zones[x].a_iWight;
		a_iHeight[x]:=zones[x].a_iHeight;
			//-
		a_iMoveX[x]:=zones[x].a_iMoveX;
		a_iMoveY[x]:=zones[x].a_iMoveY;
			//-
		a_xEnableBlocks[x]:=zones[x].a_xEnableBlocks;
		a_iSaveCurrentPosX[x]:=zones[x].a_iSaveCurrentPosX;
		a_iSaveCurrentPosY[x]:=zones[x].a_iSaveCurrentPosY;
	END_FOR
ELSIF xReloadFirstPattern THEN
	xReloadFirstPattern:=FALSE;
	FOR x:=0 TO c_iMaxZone DO
		a_sPositionRectangle[x]:=zones_FirstPattern[x].a_sPositionRectangle;
		a_iWight[x]:=zones_FirstPattern[x].a_iWight;
		a_iHeight[x]:=zones_FirstPattern[x].a_iHeight;
			//-
		a_iMoveX[x]:=zones_FirstPattern[x].a_iMoveX;
		a_iMoveY[x]:=zones_FirstPattern[x].a_iMoveY;
			//-
		a_xEnableBlocks[x]:=zones_FirstPattern[x].a_xEnableBlocks;
		a_iSaveCurrentPosX[x]:=zones_FirstPattern[x].a_iSaveCurrentPosX;
		a_iSaveCurrentPosY[x]:=zones_FirstPattern[x].a_iSaveCurrentPosY;
	END_FOR
ELSIF xReloadSecondPattern THEN
	xReloadSecondPattern:=FALSE;
	FOR x:=0 TO c_iMaxZone DO
		a_sPositionRectangle[x]:=zones_SecondPattern[x].a_sPositionRectangle;
		a_iWight[x]:=zones_SecondPattern[x].a_iWight;
		a_iHeight[x]:=zones_SecondPattern[x].a_iHeight;
			//-
		a_iMoveX[x]:=zones_SecondPattern[x].a_iMoveX;
		a_iMoveY[x]:=zones_SecondPattern[x].a_iMoveY;
			//-
		a_xEnableBlocks[x]:=zones_SecondPattern[x].a_xEnableBlocks;
		a_iSaveCurrentPosX[x]:=zones_SecondPattern[x].a_iSaveCurrentPosX;
		a_iSaveCurrentPosY[x]:=zones_SecondPattern[x].a_iSaveCurrentPosY;
	END_FOR
ELSIF xChargeEmpty THEN
	xChargeEmpty:=FALSE;
	FOR x:=0 TO c_iMaxZone DO
		a_sPositionRectangle[x]:=zones_Empty[x].a_sPositionRectangle;
		a_iWight[x]:=zones_Empty[x].a_iWight;
		a_iHeight[x]:=zones_Empty[x].a_iHeight;
			//-
		a_iMoveX[x]:=zones_Empty[x].a_iMoveX;
		a_iMoveY[x]:=zones_Empty[x].a_iMoveY;
			//-
		a_xEnableBlocks[x]:=zones_Empty[x].a_xEnableBlocks;
		a_iSaveCurrentPosX[x]:=zones_Empty[x].a_iSaveCurrentPosX;
		a_iSaveCurrentPosY[x]:=zones_Empty[x].a_iSaveCurrentPosY;
	END_FOR
END_IF

// 
// IF xSave THEN
// 	xSave:=FALSE;
// 	PersistentVars.zones_tractor[iConfSave]:=zones[iConfSave];
// ELSIF xLoad THEN
// 	xLoad:=FALSE;
// 	zones[iConfSave]:=PersistentVars.zones_tractor[iConfSave];
// END_IF
                  
END_PROGRAM

PROGRAM prg_Hmi_RobotControl2
  VAR
    sDescriptionBar : STRING(255);
    sStatusBar : STRING(255);
    sjAux : STRING;  (* - *)
    sStringJointPos : STRING;
    scAux : STRING;  (* - *)
    sStringCartPos : STRING;
    sQuaternion : STRING(255);
    lrRoll : LREAL;
    lrPitch : LREAL;
    lrYaw : LREAL;
    xToRPY : BOOL;
    rRoll : REAL;
    rPitch : REAL;
    rYaw : REAL;
    rXmm : REAL;
    rYmm : REAL;
    rZmm : REAL;
    sRPY : STRING(255);
    xIsRot : BOOL;
    arJointsInRadians : ARRAY[0..5] OF REAL;
    udiBufferSize : UDINT;
    sJointRadFormatting : STRING := '%1.3f';
    eAdapterError : IoDrvEtherNetIP.DED.ERROR;
    xDiagnosisInfoAvailable : BOOL;
    eAdapterState : IoDrvEtherNetIP.DEVICE_STATE;
    Set_IP : BOOL;
    ipDosan : ARRAY[0..3] OF BYTE;
    deinfo : IoDrvEtherNetIP.DEVICE_INFO;
    errorDE : IoDrvEtherNetIP.DED.ERROR;
    a_ipDoosan : ARRAY[0..3] OF ARRAY[0..3] OF STRING := [['192', '168', '110', '70'], 3([4('')])];
    iIndexIP : INT := 1;  (* -Default impostato sul Doosan *)
    rXMeters : REAL;
    rYMeters : REAL;
    rZMeters : REAL;
    rQW : REAL;
    rQX : REAL;
    rQY : REAL;
    rQZ : REAL;
    mR : SM3M.SMC_Matrix3;
    xComputeRotMat : BOOL;
    q : SM3M.SMC_Quat;
    sAux : STRING(255);
    iBufferSize : INT;
    sJointsInRadians : STRING(255);
  END_VAR

                    IF Set_IP THEN
	Set_IP:=FALSE;		
	ipDosan[0]:=TO_BYTE(a_ipDoosan[0][0]);
	ipDosan[1]:=TO_BYTE(a_ipDoosan[0][1]);
	ipDosan[2]:=TO_BYTE(a_ipDoosan[0][2]);
	ipDosan[3]:=TO_BYTE(a_ipDoosan[0][3]);
	DoosanRobot_EIP_Adapter_Monitoring_GPR_1.IPAddress:=ipDosan;
END_IF
errorDE:=DoosanRobot_EIP_Adapter_Monitoring_GPR_1.GetDeviceInfo(deiInfo:=deinfo);
eAdapterState := DoosanRobot_EIP_Adapter_Monitoring_GPR_1.GetDeviceState(eError => eAdapterError, xDiagnosisInfoAvailable => xDiagnosisInfoAvailable);

ACT_ConcatCartPosString();
ACT_ConcatJointPosString();

ACT_Quaternions();

ACT_JointsInRadians();











                  

ACTION ACT_ConcatJointPosString:
                        // sjAux:=TO_STRING(IO_Variables.EtherNet_IP.Joints.j1);
STU.StuSprintf(pstFormat := ADR('%3.1f'), pVarAdr := ADR(IO_Variables.g_Doosan_EIP_2.Joints.j1), udiVarType := __SYSTEM.TYPE_CLASS.TYPE_REAL, pBuffer := ADR(sjAux), dwBufferSize := udiBufferSize); 
sStringJointPos:=CONCAT(sjAux,';');

// sjAux:=TO_STRING(IO_Variables.EtherNet_IP.Joints.j2);
STU.StuSprintf(pstFormat := ADR('%3.1f'), pVarAdr := ADR(IO_Variables.g_Doosan_EIP_2.Joints.j2), udiVarType := __SYSTEM.TYPE_CLASS.TYPE_REAL, pBuffer := ADR(sjAux), dwBufferSize := udiBufferSize); 
sStringJointPos:=CONCAT(sStringJointPos,sjAux);

sjAux:=';';
sStringJointPos:=CONCAT(sStringJointPos,sjAux);

// sjAux:=TO_STRING(IO_Variables.EtherNet_IP.Joints.j3);
STU.StuSprintf(pstFormat := ADR('%3.1f'), pVarAdr := ADR(IO_Variables.g_Doosan_EIP_2.Joints.j3), udiVarType := __SYSTEM.TYPE_CLASS.TYPE_REAL, pBuffer := ADR(sjAux), dwBufferSize := udiBufferSize); 
sStringJointPos:=CONCAT(sStringJointPos,sjAux);

sjAux:=';';
sStringJointPos:=CONCAT(sStringJointPos,sjAux);

// sjAux:=TO_STRING(IO_Variables.EtherNet_IP.Joints.j4);
STU.StuSprintf(pstFormat := ADR('%3.1f'), pVarAdr := ADR(IO_Variables.g_Doosan_EIP_2.Joints.j4), udiVarType := __SYSTEM.TYPE_CLASS.TYPE_REAL, pBuffer := ADR(sjAux), dwBufferSize := udiBufferSize); 
sStringJointPos:=CONCAT(sStringJointPos,sjAux);

sjAux:=';';
sStringJointPos:=CONCAT(sStringJointPos,sjAux);

// sjAux:=TO_STRING(IO_Variables.EtherNet_IP.Joints.j5);
STU.StuSprintf(pstFormat := ADR('%3.1f'), pVarAdr := ADR(IO_Variables.g_Doosan_EIP_2.Joints.j5), udiVarType := __SYSTEM.TYPE_CLASS.TYPE_REAL, pBuffer := ADR(sjAux), dwBufferSize := udiBufferSize); 
sStringJointPos:=CONCAT(sStringJointPos,sjAux);

sjAux:=';';
sStringJointPos:=CONCAT(sStringJointPos,sjAux);

// sjAux:=TO_STRING(IO_Variables.EtherNet_IP.Joints.j6);
STU.StuSprintf(pstFormat := ADR('%3.1f'), pVarAdr := ADR(IO_Variables.g_Doosan_EIP_2.Joints.j6), udiVarType := __SYSTEM.TYPE_CLASS.TYPE_REAL, pBuffer := ADR(sjAux), dwBufferSize := udiBufferSize); 
sStringJointPos:=CONCAT(sStringJointPos,sjAux);

                      
END_ACTION

ACTION ACT_ConcatCartPosString:
                        // scAux:=TO_STRING(IO_Variables.EtherNet_IP.Cartesian.x);
STU.StuSprintf(pstFormat := ADR('%3.1f'), pVarAdr := ADR(IO_Variables.g_Doosan_EIP_2.Cartesian.x), udiVarType := __SYSTEM.TYPE_CLASS.TYPE_REAL, pBuffer := ADR(scAux), dwBufferSize := udiBufferSize); 
sStringCartPos:=CONCAT(scAux,';');

// scAux:=TO_STRING(IO_Variables.EtherNet_IP.Cartesian.y);
STU.StuSprintf(pstFormat := ADR('%3.1f'), pVarAdr := ADR(IO_Variables.g_Doosan_EIP_2.Cartesian.y), udiVarType := __SYSTEM.TYPE_CLASS.TYPE_REAL, pBuffer := ADR(scAux), dwBufferSize := udiBufferSize); 
sStringCartPos:=CONCAT(sStringCartPos,scAux);

scAux:=';';
sStringCartPos:=CONCAT(sStringCartPos,scAux);

// scAux:=TO_STRING(IO_Variables.EtherNet_IP.Cartesian.z);
STU.StuSprintf(pstFormat := ADR('%3.1f'), pVarAdr := ADR(IO_Variables.g_Doosan_EIP_2.Cartesian.z), udiVarType := __SYSTEM.TYPE_CLASS.TYPE_REAL, pBuffer := ADR(scAux), dwBufferSize := udiBufferSize); 
sStringCartPos:=CONCAT(sStringCartPos,scAux);

scAux:=';';
sStringCartPos:=CONCAT(sStringCartPos,scAux);

// scAux:=TO_STRING(IO_Variables.EtherNet_IP.Cartesian.A);
STU.StuSprintf(pstFormat := ADR('%3.1f'), pVarAdr := ADR(IO_Variables.g_Doosan_EIP_2.Cartesian.A), udiVarType := __SYSTEM.TYPE_CLASS.TYPE_REAL, pBuffer := ADR(scAux), dwBufferSize := udiBufferSize); 
sStringCartPos:=CONCAT(sStringCartPos,scAux);

scAux:=';';
sStringCartPos:=CONCAT(sStringCartPos,scAux);

// scAux:=TO_STRING(IO_Variables.EtherNet_IP.Cartesian.B);
STU.StuSprintf(pstFormat := ADR('%3.1f'), pVarAdr := ADR(IO_Variables.g_Doosan_EIP_2.Cartesian.B), udiVarType := __SYSTEM.TYPE_CLASS.TYPE_REAL, pBuffer := ADR(scAux), dwBufferSize := udiBufferSize); 
sStringCartPos:=CONCAT(sStringCartPos,scAux);

scAux:=';';
sStringCartPos:=CONCAT(sStringCartPos,scAux);

// scAux:=TO_STRING(IO_Variables.EtherNet_IP.Cartesian.C);
STU.StuSprintf(pstFormat := ADR('%3.1f'), pVarAdr := ADR(IO_Variables.g_Doosan_EIP_2.Cartesian.C), udiVarType := __SYSTEM.TYPE_CLASS.TYPE_REAL, pBuffer := ADR(scAux), dwBufferSize := udiBufferSize); 
sStringCartPos:=CONCAT(sStringCartPos,scAux);

                      
END_ACTION

ACTION ACT_Quaternions:
                        xComputeRotMat := SM3M.SMC_Matrix3_FromZYZ_deg(
	mR := mR,
	dA_deg := IO_Variables.g_Doosan_EIP_2.Cartesian.A,
	dB_deg := IO_Variables.g_Doosan_EIP_2.Cartesian.B,
	dC_deg := IO_Variables.g_Doosan_EIP_2.Cartesian.C
);

// xComputeRotMat := SM3M.SMC_Matrix3_FromRollPitchYaw_deg(
// 	mR := mR,
// 	dRoll := IO_Variables.EtherNet_IP.Cartesian.A,
// 	dPitch := IO_Variables.EtherNet_IP.Cartesian.B,
// 	dYaw := IO_Variables.EtherNet_IP.Cartesian.C
// );

xIsRot := SM3M.SMC_Matrix3_IsRotation(mR := mR, dEpsRel := 0.001);

SM3M.SMC_Quat1_From_RotMatrix(
	m := mR,
	q := q
);

xToRPY := SM3M.SMC_Matrix3_ToRollPitchYaw_deg(
	mR := mR,
	dRoll => lrRoll,
	dPitch => lrPitch,
	dYaw => lrYaw
);

/// quaternions
iBufferSize := TO_INT(XSIZEOF(sQuaternion));
sQuaternion := '';

// ROUND

rXmm := TO_REAL(IO_Variables.g_Doosan_EIP_2.Cartesian.x);
rYmm := TO_REAL(IO_Variables.g_Doosan_EIP_2.Cartesian.y);
rZmm := TO_REAL(IO_Variables.g_Doosan_EIP_2.Cartesian.z);

rXMeters := rXmm / 1000.0;
rYMeters := rYmm / 1000.0;
rZMeters := rZmm / 1000.0;

// rQW := TO_REAL(TO_INT(q.dR * 1E6)) / 1E6;
// rQX := TO_REAL(TO_INT(q.dI * 1E6)) / 1E6;
// rQY := TO_REAL(TO_INT(q.dJ * 1E6)) / 1E6;
// rQZ := TO_REAL(TO_INT(q.dK * 1E6)) / 1E6;
rQW := TO_REAL(q.dR);
rQX := TO_REAL(q.dI);
rQY := TO_REAL(q.dJ);
rQZ := TO_REAL(q.dK);

rRoll := TO_REAL(lrRoll);
rPitch := TO_REAL(lrPitch);
rYaw := TO_REAL(lrYaw);

// QUATERNION
sAux := ''; //X
STU.StuSprintf(pstFormat := ADR('%1.3f'), pVarAdr := ADR(rXMeters), udiVarType := __SYSTEM.TYPE_CLASS.TYPE_REAL, pBuffer := ADR(sAux), dwBufferSize := udiBufferSize); 
// sAux := TO_STRING(rXMeters);
STU.StrConcatA(pstTo := ADR(sQuaternion), pstFrom := ADR(sAux), iBufferSize := iBufferSize);

STU.StrConcatA(pstTo := ADR(sQuaternion), pstFrom := ADR(';'), iBufferSize := iBufferSize);

sAux := ''; //Y
STU.StuSprintf(pstFormat := ADR('%1.3f'), pVarAdr := ADR(rYMeters), udiVarType := __SYSTEM.TYPE_CLASS.TYPE_REAL, pBuffer := ADR(sAux), dwBufferSize := udiBufferSize); 
// sAux := TO_STRING(rYMeters);
STU.StrConcatA(pstTo := ADR(sQuaternion), pstFrom := ADR(sAux), iBufferSize := iBufferSize);

STU.StrConcatA(pstTo := ADR(sQuaternion), pstFrom := ADR(';'), iBufferSize := iBufferSize);

sAux := ''; //Z
STU.StuSprintf(pstFormat := ADR('%1.3f'), pVarAdr := ADR(rZMeters), udiVarType := __SYSTEM.TYPE_CLASS.TYPE_REAL, pBuffer := ADR(sAux), dwBufferSize := udiBufferSize);
// sAux := TO_STRING(rZMeters);
STU.StrConcatA(pstTo := ADR(sQuaternion), pstFrom := ADR(sAux), iBufferSize := iBufferSize);

STU.StrConcatA(pstTo := ADR(sQuaternion), pstFrom := ADR(';'), iBufferSize := iBufferSize);

sAux := ''; //qx
STU.StuSprintf(pstFormat := ADR('%1.3f'), pVarAdr := ADR(rQX), udiVarType := __SYSTEM.TYPE_CLASS.TYPE_REAL, pBuffer := ADR(sAux), dwBufferSize := udiBufferSize);
// sAux := TO_STRING(rQX);
STU.StrConcatA(pstTo := ADR(sQuaternion), pstFrom := ADR(sAux), iBufferSize := iBufferSize);

STU.StrConcatA(pstTo := ADR(sQuaternion), pstFrom := ADR(';'), iBufferSize := iBufferSize);

sAux := ''; //qy
STU.StuSprintf(pstFormat := ADR('%1.3f'), pVarAdr := ADR(rQY), udiVarType := __SYSTEM.TYPE_CLASS.TYPE_REAL, pBuffer := ADR(sAux), dwBufferSize := udiBufferSize);
// sAux := TO_STRING(rQY);
STU.StrConcatA(pstTo := ADR(sQuaternion), pstFrom := ADR(sAux), iBufferSize := iBufferSize);

STU.StrConcatA(pstTo := ADR(sQuaternion), pstFrom := ADR(';'), iBufferSize := iBufferSize);

sAux := ''; //qz
STU.StuSprintf(pstFormat := ADR('%1.3f'), pVarAdr := ADR(rQZ), udiVarType := __SYSTEM.TYPE_CLASS.TYPE_REAL, pBuffer := ADR(sAux), dwBufferSize := udiBufferSize);
// sAux := TO_STRING(rQZ);
STU.StrConcatA(pstTo := ADR(sQuaternion), pstFrom := ADR(sAux), iBufferSize := iBufferSize);

STU.StrConcatA(pstTo := ADR(sQuaternion), pstFrom := ADR(';'), iBufferSize := iBufferSize);

sAux := ''; //qw
STU.StuSprintf(pstFormat := ADR('%1.3f'), pVarAdr := ADR(rQW), udiVarType := __SYSTEM.TYPE_CLASS.TYPE_REAL, pBuffer := ADR(sAux), dwBufferSize := udiBufferSize);
// sAux := TO_STRING(rQW);
STU.StrConcatA(pstTo := ADR(sQuaternion), pstFrom := ADR(sAux), iBufferSize := iBufferSize);

(*----------------------------------------------*)
// RPY
iBufferSize := TO_INT(XSIZEOF(sRPY));
sRPY := '';

sAux := ''; //X
STU.StuSprintf(pstFormat := ADR('%5.1f'), pVarAdr := ADR(rXmm), udiVarType := __SYSTEM.TYPE_CLASS.TYPE_REAL, pBuffer := ADR(sAux), dwBufferSize := udiBufferSize);
// sAux := TO_STRING(rXmm);
STU.StrConcatA(pstTo := ADR(sRPY), pstFrom := ADR(sAux), iBufferSize := iBufferSize);

STU.StrConcatA(pstTo := ADR(sRPY), pstFrom := ADR(';'), iBufferSize := iBufferSize);

sAux := ''; //Y
STU.StuSprintf(pstFormat := ADR('%5.1f'), pVarAdr := ADR(rYmm), udiVarType := __SYSTEM.TYPE_CLASS.TYPE_REAL, pBuffer := ADR(sAux), dwBufferSize := udiBufferSize);
// sAux := TO_STRING(rYmm);
STU.StrConcatA(pstTo := ADR(sRPY), pstFrom := ADR(sAux), iBufferSize := iBufferSize);

STU.StrConcatA(pstTo := ADR(sRPY), pstFrom := ADR(';'), iBufferSize := iBufferSize);

sAux := ''; //Z
STU.StuSprintf(pstFormat := ADR('%5.1f'), pVarAdr := ADR(rZmm), udiVarType := __SYSTEM.TYPE_CLASS.TYPE_REAL, pBuffer := ADR(sAux), dwBufferSize := udiBufferSize);
// sAux := TO_STRING(rZmm);
STU.StrConcatA(pstTo := ADR(sRPY), pstFrom := ADR(sAux), iBufferSize := iBufferSize);

STU.StrConcatA(pstTo := ADR(sRPY), pstFrom := ADR(';'), iBufferSize := iBufferSize);

sAux := ''; //roll
STU.StuSprintf(pstFormat := ADR('%3.1f'), pVarAdr := ADR(rRoll), udiVarType := __SYSTEM.TYPE_CLASS.TYPE_REAL, pBuffer := ADR(sAux), dwBufferSize := udiBufferSize);
// sAux := TO_STRING(rRoll);
STU.StrConcatA(pstTo := ADR(sRPY), pstFrom := ADR(sAux), iBufferSize := iBufferSize);

STU.StrConcatA(pstTo := ADR(sRPY), pstFrom := ADR(';'), iBufferSize := iBufferSize);

sAux := ''; //pitch
STU.StuSprintf(pstFormat := ADR('%3.1f'), pVarAdr := ADR(rPitch), udiVarType := __SYSTEM.TYPE_CLASS.TYPE_REAL, pBuffer := ADR(sAux), dwBufferSize := udiBufferSize);
// sAux := TO_STRING(rPitch);
STU.StrConcatA(pstTo := ADR(sRPY), pstFrom := ADR(sAux), iBufferSize := iBufferSize);

STU.StrConcatA(pstTo := ADR(sRPY), pstFrom := ADR(';'), iBufferSize := iBufferSize);

sAux := ''; //yaw
STU.StuSprintf(pstFormat := ADR('%3.1f'), pVarAdr := ADR(rYaw), udiVarType := __SYSTEM.TYPE_CLASS.TYPE_REAL, pBuffer := ADR(sAux), dwBufferSize := udiBufferSize);
// sAux := TO_STRING(rYaw);
STU.StrConcatA(pstTo := ADR(sRPY), pstFrom := ADR(sAux), iBufferSize := iBufferSize);

                      
END_ACTION

ACTION ACT_JointsInRadians:
                        arJointsInRadians[0] := IO_Variables.g_Doosan_EIP_2.Joints.j1 * TO_REAL(SMC_FACTOR_DEG_TO_RAD);
arJointsInRadians[1] := IO_Variables.g_Doosan_EIP_2.Joints.j2 * TO_REAL(SMC_FACTOR_DEG_TO_RAD);
arJointsInRadians[2] := IO_Variables.g_Doosan_EIP_2.Joints.j3 * TO_REAL(SMC_FACTOR_DEG_TO_RAD);
arJointsInRadians[3] := IO_Variables.g_Doosan_EIP_2.Joints.j4 * TO_REAL(SMC_FACTOR_DEG_TO_RAD);
arJointsInRadians[4] := IO_Variables.g_Doosan_EIP_2.Joints.j5 * TO_REAL(SMC_FACTOR_DEG_TO_RAD);
arJointsInRadians[5] := IO_Variables.g_Doosan_EIP_2.Joints.j6 * TO_REAL(SMC_FACTOR_DEG_TO_RAD);


(*----------------------------------------------*)
// Radians
iBufferSize := TO_INT(XSIZEOF(sJointsInRadians));
udiBufferSize := TO_UDINT(XSIZEOF(sJointsInRadians));
sJointsInRadians := '';

sAux := ''; // j1
STU.StuSprintf(pstFormat := ADR('%1.3f'), pVarAdr := ADR(arJointsInRadians[0]), udiVarType := __SYSTEM.TYPE_CLASS.TYPE_REAL, pBuffer := ADR(sAux), dwBufferSize := udiBufferSize); 
// sAux := TO_STRING(arJointsInRadians[0]);
STU.StrConcatA(pstTo := ADR(sJointsInRadians), pstFrom := ADR(sAux), iBufferSize := iBufferSize);

STU.StrConcatA(pstTo := ADR(sJointsInRadians), pstFrom := ADR(';'), iBufferSize := iBufferSize);

sAux := ''; // j2
STU.StuSprintf(pstFormat := ADR('%1.3f'), pVarAdr := ADR(arJointsInRadians[1]), udiVarType := __SYSTEM.TYPE_CLASS.TYPE_REAL, pBuffer := ADR(sAux), dwBufferSize := udiBufferSize); 
// sAux := TO_STRING(arJointsInRadians[1]);
STU.StrConcatA(pstTo := ADR(sJointsInRadians), pstFrom := ADR(sAux), iBufferSize := iBufferSize);

STU.StrConcatA(pstTo := ADR(sJointsInRadians), pstFrom := ADR(';'), iBufferSize := iBufferSize);

sAux := ''; //j3
STU.StuSprintf(pstFormat := ADR('%1.3f'), pVarAdr := ADR(arJointsInRadians[2]), udiVarType := __SYSTEM.TYPE_CLASS.TYPE_REAL, pBuffer := ADR(sAux), dwBufferSize := udiBufferSize); 
// sAux := TO_STRING(arJointsInRadians[2]);
STU.StrConcatA(pstTo := ADR(sJointsInRadians), pstFrom := ADR(sAux), iBufferSize := iBufferSize);

STU.StrConcatA(pstTo := ADR(sJointsInRadians), pstFrom := ADR(';'), iBufferSize := iBufferSize);

sAux := ''; //j4
STU.StuSprintf(pstFormat := ADR('%1.3f'), pVarAdr := ADR(arJointsInRadians[3]), udiVarType := __SYSTEM.TYPE_CLASS.TYPE_REAL, pBuffer := ADR(sAux), dwBufferSize := udiBufferSize); 
// sAux := TO_STRING(arJointsInRadians[3]);
STU.StrConcatA(pstTo := ADR(sJointsInRadians), pstFrom := ADR(sAux), iBufferSize := iBufferSize);

STU.StrConcatA(pstTo := ADR(sJointsInRadians), pstFrom := ADR(';'), iBufferSize := iBufferSize);

sAux := ''; //j5
STU.StuSprintf(pstFormat := ADR('%1.3f'), pVarAdr := ADR(arJointsInRadians[4]), udiVarType := __SYSTEM.TYPE_CLASS.TYPE_REAL, pBuffer := ADR(sAux), dwBufferSize := udiBufferSize); 
// sAux := TO_STRING(arJointsInRadians[4]);
STU.StrConcatA(pstTo := ADR(sJointsInRadians), pstFrom := ADR(sAux), iBufferSize := iBufferSize);

STU.StrConcatA(pstTo := ADR(sJointsInRadians), pstFrom := ADR(';'), iBufferSize := iBufferSize);

sAux := ''; //j6
STU.StuSprintf(pstFormat := ADR('%1.3f'), pVarAdr := ADR(arJointsInRadians[5]), udiVarType := __SYSTEM.TYPE_CLASS.TYPE_REAL, pBuffer := ADR(sAux), dwBufferSize := udiBufferSize); 
// sAux := TO_STRING(arJointsInRadians[5]);
STU.StrConcatA(pstTo := ADR(sJointsInRadians), pstFrom := ADR(sAux), iBufferSize := iBufferSize);
                      
END_ACTION
END_PROGRAM

